// Internal/Blocks/GetStatusMessage
(* ===============================================================================
   FESTO AG & Co. KG, Esslingen - Copyright 2015. All rights reserved.                       
 ---------------------------------------------------------------------------------
 Functionblock:  GetStatusMessage 
 Description:    function to get discription of the status of function block or FPC 
 Version:        V 1.0        
 Composer:       Benjamin Kilgus
 Last Update:    10.04.2014                                                                          
------------------------------------------------------------------------------- *)
{library private}
(* ----------------------------------------------------------------------------
Date        Name            	Activity                                                                              
10.04.2014	Benjamin Kilgus     created
=============================================================================== *)
{library public}

FUNCTION GetStatusMessage : STRING

VAR_INPUT
  StatusIn   	: DT_FML_STATUS;
END_VAR

VAR
  StatusStringCat  	: STRING;
  StatusStringID  	: STRING;
END_VAR

(* ===== logic part ================================================= *)
 // get category string 
 CASE StatusIn.Cat OF
	 
 	FML_no_category:
		StatusStringCat := '';
		// get ID string 
		CASE StatusIn.ID OF
			 0:     StatusStringID := 'no error';
			 ELSE   StatusStringID := 'unknown number';
		END_CASE

		 
	FML_function_block:	
		StatusStringCat := 'FB: ';
		// get ID string 
	  	CASE StatusIn.ID OF
			 0:     StatusStringID := 'no error';
			 1:     StatusStringID := 'initialization is active';
			 2:     StatusStringID := 'function block is busy';
			10:     StatusStringID := 'other FPC function block is active';
			20:     StatusStringID := 'timeout of function block';
			30:     StatusStringID := 'device type is not valid';
			40:     StatusStringID := 'wrong access value';
			50:     StatusStringID := 'pointer to zero';
			51:     StatusStringID := 'pointer wrong size';
			60:     StatusStringID := 'FHPP+ data configuration not valid';
			ELSE 	StatusStringID := 'unknown number';
		END_CASE
		
		
	FML_reserved:
		StatusStringCat := 'reserved: ';

	FML_parameter_transfer:
		StatusStringCat	:= 'FPC: ';
		// get ID string 
	  	CASE StatusIn.ID OF
			 0:      StatusStringID := 'non-permitted PNU';
			 1:      StatusStringID := 'parameter is read only';
			 2:      StatusStringID := 'lower or upper limit value exceeded';
			 3:      StatusStringID := 'wrong subindex';
			 4:      StatusStringID := 'no array';
			 5:      StatusStringID := 'incorrect data type';
			 6:      StatusStringID := 'setting not permitted (only reset allowed)';
			 7:      StatusStringID := 'describing element cannot be modified';
			 8:      StatusStringID := 'PPO-Write requested in IR does not exist';
			 9:      StatusStringID := 'description data do not exist';
			10:      StatusStringID := 'access group incorrect';
			11:      StatusStringID := 'no control rights';
			12:      StatusStringID := 'password incorrect';
			13:      StatusStringID := 'text not readable in cyclic exchange';
			14:      StatusStringID := 'name not readable in cyclic exchange';
			15:      StatusStringID := 'text array does not exist';
			16:      StatusStringID := 'PPO-Write missing';
			17:      StatusStringID := 'order cannot be processed because of operating status';
			18:      StatusStringID := 'other Errors';
			19:      StatusStringID := 'date not readable in cyclic exchange';
			20:      StatusStringID := 'non-permitted value';
			22:      StatusStringID := 'non-permitted Attributes, number of elements, PNU or IND';
			23:      StatusStringID := 'write request: non-permitted format';
			24:      StatusStringID := 'write request: Number of values not permitted';
			25..100: StatusStringID := 'reserved for PROFIBUS';
			101:     StatusStringID := 'ReqID is not supported';
			102:     StatusStringID := 'parameter is write only';
			103..255:StatusStringID := 'reserved for Festo';
			
			//FILETRANSFER
			1001: 	StatusStringID := 'wrong sequence number';
			1002: 	StatusStringID := 'timeout between two packets';
			1003: 	StatusStringID := 'wrong packet format';
			1004: 	StatusStringID := 'false instruction';
			1005: 	StatusStringID := 'read error';
			1006:	StatusStringID := 'write error';
			1007:	StatusStringID := 'data volume is not correct';
			1008: 	StatusStringID := 'parameterfile error';
			1009: 	StatusStringID := 'fault not receipt';
			1010: 	StatusStringID := 'timeout';
			1011: 	StatusStringID := 'file open error';
			1012: 	StatusStringID := 'file close error';
			1013: 	StatusStringID := 'file delete error';
			1014: 	StatusStringID := 'directory create error';
			1015: 	StatusStringID := 'file not exist';
			1016: 	StatusStringID := 'file read error';
			1017: 	StatusStringID := 'get size error';
			1018: 	StatusStringID := 'file write error';
			1019:	StatusStringID := 'no or double direction selected';
			1020:	StatusStringID := 'filename is empty';
			1021:	StatusStringID := 'size of parameterfile too short/long';
			1022:	StatusStringID := 'parameterfile is not complete';
			
			ELSE 	StatusStringID := 'unknown number';
		END_CASE
			
	ELSE
		StatusStringCat := 'unknown status category';
 END_CASE

 
 GetStatusMessage := CONCAT(StatusStringCat, StatusStringID);  // Return the resulting string
 
(* ===== end of function ================================== *)

END_FUNCTION

// Blocks/FML_Read
(* ============================================================================
   FESTO AG & Co. KG, Esslingen - Copyright (c) 2015. All rights reserved.                       

 Functionblock:  FML_Read
 Description:    function block to read the input data from the controller
 Version:        V3.5.7.21        
 Composer:       chmm
 Date:           13.11.2017                                                                          
------------------------------------------------------------------------------- *)
{library private}
(* ----------------------------------------------------------------------------
Date        Name             	Activity                                                                              
22.06.2015	Christian Hammer	created
13.11.2017	Christian Hammer	added SFC-DC and MTR-DCI controller
=============================================================================== *)
{library public}


FUNCTION_BLOCK FML_Read

VAR_IN_OUT
	FML_REF					: DT_FML_REF; 						// structure of the parameter to control and parametrize the motorcontroller
END_VAR

VAR_INPUT
	DeviceType				: E_FML_DEVICE_TYPE; 				// type of the controller
	Modbus					: BOOL;								// 1 = modbus is using / 0 = other fieldbus is using
	HighByteFirst			: BOOL;								// byteorder (1 = high byte first)
	FPC_active				: BOOL;								// ParameterChannel (FPC) in use
	PlcConfigFHPP_PLUS_IN	: UDINT;							// plc configuration code (is displayed in the Festo Configuration Tool (FCT))
	
	FHPP_Source				: ARRAY [0..7] OF BYTE;				// input FHPP Data (from controller)
	FPC_Source				: ARRAY [0..7] OF BYTE;				// input FPC Data (from controller)
	FHPP_PLUS_Source1		: ARRAY [0..7] OF BYTE;				// first 8 bytes of FHPP+ input data (from controller)
	FHPP_PLUS_Source2		: ARRAY [0..7] OF BYTE;				// second 8 bytes of FHPP+ input data (from controller)
	FHPP_PLUS_Source3		: ARRAY [0..7] OF BYTE;				// third 8 bytes of FHPP+ input data (from controller)
END_VAR

VAR_OUTPUT
	Error					: BOOL;								// transmission fault
	Status          		: DT_FML_STATUS;     				// return value of function block
END_VAR

VAR
	FHPP_Read				: FHPP_Read;						// function block read FHPP data
	FPC_Read				: FPC_Read;							// function block read FPC data
	FHPP_PLUS_Read			: FHPP_PLUS_Read;					// function block read FHPP+ data
END_VAR

// function block (FB) is busy
Status.Err:=FALSE; Status.Cat:=FML_function_block; Status.ID:=FML_fb_busy;

// check and set DeviceType of the controller
IF DeviceType = CMMO_ST OR DeviceType = EMCA_EC OR DeviceType = CMMP_AS OR DeviceType = CMMS_AS OR DeviceType = CMMS_ST OR DeviceType = CMMD_AS OR DeviceType = SFC_DC OR DeviceType = MTR_DCI THEN  
	FML_REF.DeviceType	:= DeviceType;
ELSE
	Status.Err:=TRUE; Status.Cat:=FML_function_block; Status.ID:=FML_wrong_device;
END_IF

// set type of bus and byteorder
FML_REF.Modbus			:= Modbus;
FML_REF.HighByteFirst	:= HighByteFirst;

// mode of the parameter channel (in use or not)
FML_REF.FPC_active		:= FPC_active;

// reading and mapping of FHPP bus data 
FHPP_Read(
	FML_REF				:= FML_REF,
	FHPP_Source			:= FHPP_Source);
		
// if parameter-channel (FPC) is activated - reading and mapping of FPC bus data	
IF FML_REF.FPC_active THEN
	FPC_Read(
		FML_REF			:= FML_REF,
		FPC_Source		:= FPC_Source);
END_IF

IF (PlcConfigFHPP_PLUS_IN<>0) AND (Status.Err = FALSE) THEN
	FHPP_PLUS_Read(
		FML_REF					:= FML_REF,
		PlcConfigFHPP_PLUS_IN	:= PlcConfigFHPP_PLUS_IN,
		FHPP_PLUS_Source1		:= FHPP_PLUS_Source1,
		FHPP_PLUS_Source2		:= FHPP_PLUS_Source2,
		FHPP_PLUS_Source3		:= FHPP_PLUS_Source3,
		Status					=> Status);		
END_IF	
	
IF (Status.Err = FALSE) THEN
	// reading done - no error
	Status.Err:=FALSE; Status.Cat:=FML_no_category; Status.ID:=FML_no_error;
END_IF	

Status.Msg						:= GetStatusMessage(Status);
Error							:= Status.Err;

(* ===== end of function block ============================= *)

END_FUNCTION_BLOCK

// Internal/Blocks/ReadWriteData/FHPP_Read
(* ===============================================================================
   FESTO AG & Co. KG, Esslingen - Copyright 2015. All rights reserved.                       
 ---------------------------------------------------------------------------------
 Functionblock:  FHPP_Read  
 Description:    function block to read an mapp the FHPP data from the controller
 Version:        V 3.5.4.4        
 Composer:       chmm 
 Last Update:    22.06.2015                                                                           
------------------------------------------------------------------------------- *)
{library private}
(* ----------------------------------------------------------------------------
Date        Name            	Activity                                                                              
22.06.2015	Christian Hammer	created
=============================================================================== *)
{library public}

FUNCTION_BLOCK FHPP_Read

VAR_IN_OUT
	FML_REF			: DT_FML_REF;						// structure of the parameter to control and parametrize the motorcontroller
END_VAR

VAR_INPUT
	FHPP_Source		: ARRAY [0..7] OF BYTE;				// input FHPP data (from controller)
END_VAR

VAR
	pFHPP_DATA_IN	: POINTER TO ARRAY[0..7] OF BYTE;	// pointer to FHPP data
END_VAR

(***********************************************************************************************************************************************
*********** INPUT FHPP DATA ********************************************************************************************************************
***********************************************************************************************************************************************)

pFHPP_DATA_IN				:= ADR(FML_REF.FHPP.IN);

IF FML_REF.Modbus THEN				// modbus word swapping
	pFHPP_DATA_IN^[0]		:= FHPP_Source[1]; 
	pFHPP_DATA_IN^[1]		:= FHPP_Source[0]; 
	pFHPP_DATA_IN^[2]		:= FHPP_Source[3]; 
	pFHPP_DATA_IN^[3]		:= FHPP_Source[2];
	IF FML_REF.HighByteFirst THEN	// high byte first (actual value2)
		pFHPP_DATA_IN^[4]	:= FHPP_Source[6]; 
		pFHPP_DATA_IN^[5] 	:= FHPP_Source[7]; 
		pFHPP_DATA_IN^[6] 	:= FHPP_Source[4]; 
		pFHPP_DATA_IN^[7] 	:= FHPP_Source[5];
	ELSE							// low byte first (actual value2)
		pFHPP_DATA_IN^[4]	:= FHPP_Source[5]; 
		pFHPP_DATA_IN^[5] 	:= FHPP_Source[4]; 
		pFHPP_DATA_IN^[6] 	:= FHPP_Source[7]; 
		pFHPP_DATA_IN^[7] 	:= FHPP_Source[6];
	END_IF

ELSE								// normal fieldbus: copy only
	pFHPP_DATA_IN^[0]		:= FHPP_Source[0]; 
	pFHPP_DATA_IN^[1]		:= FHPP_Source[1]; 
	pFHPP_DATA_IN^[2]		:= FHPP_Source[2]; 
	pFHPP_DATA_IN^[3]		:= FHPP_Source[3]; 
	IF FML_REF.HighByteFirst THEN	// high byte first (actual value2)
		pFHPP_DATA_IN^[4]	:= FHPP_Source[7]; 
		pFHPP_DATA_IN^[5] 	:= FHPP_Source[6]; 
		pFHPP_DATA_IN^[6] 	:= FHPP_Source[5]; 
		pFHPP_DATA_IN^[7] 	:= FHPP_Source[4];
	ELSE							// low byte first (actual value2)
		pFHPP_DATA_IN^[4]	:= FHPP_Source[4]; 
		pFHPP_DATA_IN^[5] 	:= FHPP_Source[5]; 
		pFHPP_DATA_IN^[6] 	:= FHPP_Source[6]; 
		pFHPP_DATA_IN^[7] 	:= FHPP_Source[7];
	END_IF
END_IF

(* ===== end of function block ============================= *)

END_FUNCTION_BLOCK

// Internal/Blocks/ReadWriteData/FPC_Read
(* ===============================================================================
   FESTO AG & Co. KG, Esslingen - Copyright 2015. All rights reserved.                       
 ---------------------------------------------------------------------------------
 Functionblock:  FPC_Read  
 Description:    function block to read an mapp the FPC data from the controller
 Version:        V 3.5.7.21        
 Composer:       chmm 
 Last Update:    20.11.2017                                                                           
------------------------------------------------------------------------------- *)
{library private}
(* ----------------------------------------------------------------------------
Date        Name            	Activity                                                                              
22.06.2015	Christian Hammer	created
20.11.2017	Christian Hammer	ResponseID´s for SFC-DC and MTR-DCI added
=============================================================================== *)
{library public}

FUNCTION_BLOCK FPC_Read

VAR_IN_OUT
	FML_REF			: DT_FML_REF;						// structure of the parameter to control and parametrize the motorcontroller
END_VAR	

VAR_INPUT
	FPC_Source		: ARRAY [0..7] OF BYTE;				// input FPC data (from controller)
END_VAR

VAR
	pFPC_DATA_IN	: POINTER TO ARRAY[0..7] OF BYTE;	// pointer to FPC data
	pFML_Ref_FPC_In	: POINTER TO ARRAY[0..7] OF BYTE;	// pointer to FML-Ref-FPC.In for copying paramter files or firmware files
	RespID			: INT;
END_VAR

(***********************************************************************************************************************************************
*********** INPUT FPC DATA *********************************************************************************************************************
***********************************************************************************************************************************************)

pFPC_DATA_IN				:= ADR(FML_REF.FPC.IN);

IF FML_REF.Modbus THEN				// modbus word swapping
	pFPC_DATA_IN^[0]		:= FPC_Source[1]; 
	pFPC_DATA_IN^[1]		:= FPC_Source[0]; 
	IF FML_REF.HighByteFirst THEN	// high bytes first (ParID and value)
		pFPC_DATA_IN^[2]	:= FPC_Source[2]; 
		pFPC_DATA_IN^[3]	:= FPC_Source[3];
		pFPC_DATA_IN^[4]	:= FPC_Source[6]; 
		pFPC_DATA_IN^[5] 	:= FPC_Source[7]; 
		pFPC_DATA_IN^[6] 	:= FPC_Source[4]; 
		pFPC_DATA_IN^[7] 	:= FPC_Source[5];
	ELSE							// low bytes first (ParID and value)
		pFPC_DATA_IN^[2]	:= FPC_Source[3]; 
		pFPC_DATA_IN^[3]	:= FPC_Source[2];
		pFPC_DATA_IN^[4]	:= FPC_Source[5]; 
		pFPC_DATA_IN^[5] 	:= FPC_Source[4]; 
		pFPC_DATA_IN^[6] 	:= FPC_Source[7]; 
		pFPC_DATA_IN^[7] 	:= FPC_Source[6];
	END_IF

ELSE								//normal fieldbus: copy only
	pFPC_DATA_IN^[0]		:= FPC_Source[0]; 
	pFPC_DATA_IN^[1]		:= FPC_Source[1];
	IF FML_REF.HighByteFirst THEN	// high byte first (ParID and value)
		pFPC_DATA_IN^[2]	:= FPC_Source[3]; 
		pFPC_DATA_IN^[3]	:= FPC_Source[2];
		pFPC_DATA_IN^[4]	:= FPC_Source[7]; 
		pFPC_DATA_IN^[5] 	:= FPC_Source[6]; 
		pFPC_DATA_IN^[6] 	:= FPC_Source[5]; 
		pFPC_DATA_IN^[7] 	:= FPC_Source[4];	
	ELSE 							// low bytes first (ParID and value)
		pFPC_DATA_IN^[2]	:= FPC_Source[2]; 
		pFPC_DATA_IN^[3]	:= FPC_Source[3];
		pFPC_DATA_IN^[4]	:= FPC_Source[4]; 
		pFPC_DATA_IN^[5] 	:= FPC_Source[5]; 
		pFPC_DATA_IN^[6] 	:= FPC_Source[6]; 
		pFPC_DATA_IN^[7] 	:= FPC_Source[7];
	END_IF	
END_IF



(*-----------------------------------------------------------
     assignment of the input data (stateword)
------------------------------------------------------------*)
(* byte 1 FPCS *)
FML_REF.FPCS_Modus 				:= SHR((FML_REF.FPC.IN.ModeAK AND 2#11110000),4);

(*-----------------------------------------------------------
     decoding of EFPC modus
------------------------------------------------------------*)
CASE FML_REF.FPCS_Modus OF
	1,2,3:(* FPCS_Modus 1=PNU extended; 2= internal data object; 3=CAN objects *)

	(*
	|-------- byte 1 ------|- byte 2 -|---------- byte 3..4 ------------------------|- byte 5..8 -|
	| 7  6  5  4 | 3 2 1 0 |          | 15 14 ..                 			 .. 1 0 |             |
	| FPCS mode	 |   AK    | subindex | PNU extended or data object or CAN object	|    value    |
	-----------------------------------------------------------------------------------------------		
		AK:  request identifier (Auftragskennung) *)			
		
		FML_REF.RespID	 		:= (FML_REF.FPC.IN.ModeAK AND 2#00001111);		// FPCS mode (byte 1)	
		FML_REF.ActSubindex 	:= FML_REF.FPC.IN.IND;   						// save subindex (byte 2)		
		FML_REF.ActValue		:= FML_REF.FPC.IN.Value; 						// parameter value (byte 5..8)
		FML_REF.ActPNU 			:= FML_REF.FPC.IN.ParID;						// **PKE/ PNU/ data object/ CAN (byte 3+4)

	4,5:(* FPCS_Modus 4=parameter file; 5=firmware file 
      	|------ byte 1 -----------|-- byte 2 -|--byte 3..8 -----|
	    | 7  6  5  4 | 3  2  1  0 |           | 				|
	    | FPCS Modus |   res      | Packet-ID |  6 Byte Data	|
	    -------------------------------------------------------		
		  packet-ID: -------------- byte 2 ----------
		             | 7    6    5  | 4  3  2  1  0 |
		             | control bits |   sequence-nr |
		             -------------------------------- *)		
		//---- FPCS mode (byte 1) ---- 
		FML_REF.RespID						:= (FML_REF.FPC.IN.ModeAK AND 2#00001111);
		//---- byte 2 packet-ID ----	
		FML_REF.FPCS_Packet.BitSequenceNr 	:= (FML_REF.FPC.IN.IND AND 2#00011111);
		FML_REF.FPCS_Packet.Control			:= SHR((FML_REF.FPC.IN.IND AND 2#11100000),5);
		//---- byte 3..8 data ----	
		pFML_Ref_FPC_In						:= ADR(FML_REF.FPC.IN);			// byte swapping for modbus data
		FML_REF.FPCS_Packet.Data[1]			:= pFML_Ref_FPC_In^[3];  
		FML_REF.FPCS_Packet.Data[2] 		:= pFML_Ref_FPC_In^[2];  
		FML_REF.FPCS_Packet.Data[3] 		:= pFML_Ref_FPC_In^[7];  
		FML_REF.FPCS_Packet.Data[4] 		:= pFML_Ref_FPC_In^[6];  
		FML_REF.FPCS_Packet.Data[5] 		:= pFML_Ref_FPC_In^[5];  
		FML_REF.FPCS_Packet.Data[6] 		:= pFML_Ref_FPC_In^[4]; 
	
	ELSE  (* FPCS_Modus = standard ----
  		|-byte 1 -|- byte 2 -|---------------- byte 3 --------------|- byte 5..8 -|
		|         |          |15 14 13 12| 11|10 9 8 7 6 5 4 3 2 1 0|             |
		|   res   | subindex |     AK    |SPM|        PNU           |   value     |
		---------------------------------------------------------------------------		
			byte 1: reserved
			byte 2: subindex
			AK:     response identifier (Antwortkennung)
			SPM:    NOT used
			PNU:    Parameternummer / parametern umber *)				

		FML_REF.ActSubindex 	:= FML_REF.FPC.IN.IND;  	 // save subindex
		
		(* Byte 3+4 **PKE/ PNU/ data object/ CAN** *)
		FML_REF.ActValue		:= FML_REF.FPC.IN.Value;
		RespID					:= WORD_TO_INT( SHR((INT_TO_WORD(FML_REF.FPC.IN.ParID) AND 2#1111000000000000),12));
		FML_REF.RespID			:= RespID;
		FML_REF.ActPNU 			:= WORD_TO_INT( INT_TO_WORD(FML_REF.FPC.IN.ParID) AND 2#0000011111111111);
		
		(* Byte 5..8 parameter value *)
END_CASE

CASE FML_REF.RespID OF
	
	 0,3:(* No instruction or transmission is activ *)
		FML_REF.Done            := FALSE;
		FML_REF.Err             := FALSE;
		FML_REF.DatatypeRD      := 0;
		FML_REF.ActPNU          := 0;
		FML_REF.ActSubindex     := 0;
		FML_REF.ActValue    	:= 0;
			
	1,4:(* WORD Parameter transmitted *)
		FML_REF.Done            := TRUE;
		FML_REF.Err             := FALSE;
		FML_REF.DatatypeRD      := 2;
	
	2,5:(* DWORD Parameter transmitted *)
		FML_REF.Done            := TRUE;
		FML_REF.Err             := FALSE;
		FML_REF.DatatypeRD      := 4;
			
	7:(* Transmission Err *)
		FML_REF.Done            := TRUE;
		FML_REF.Err             := TRUE;
		FML_REF.DatatypeRD      := 0;
			
	11,12:(* BYTE Parameter transmitted *)
		FML_REF.Done            := TRUE;
		FML_REF.Err             := FALSE;
		FML_REF.DatatypeRD      := 1;
		
	ELSE (* not specified*)
		FML_REF.Done        	:= TRUE;
		FML_REF.Err           	:= TRUE;
		FML_REF.DatatypeRD      := 0;	
END_CASE

(* ===== end of function block ============================= *)

END_FUNCTION_BLOCK

// Blocks/FML_Write
(* ============================================================================
   FESTO AG & Co. KG, Esslingen - Copyright (c) 2015. All rights reserved.                       

 Functionblock:  FML_Write
 Description:    function block to write the output data to the controller
 Version:        V3.5.4.4        
 Composer:       chmm
 Date:           04.09.2015                                                                           
------------------------------------------------------------------------------- *)
{library private}
(* ----------------------------------------------------------------------------
Date        Name             	Activity                                                                              
22.06.2015	Christian Hammer	created	
=============================================================================== *)
{library public}

FUNCTION_BLOCK FML_Write

VAR_IN_OUT
	FML_REF					: DT_FML_REF; 
END_VAR

VAR_INPUT
	PlcConfigFHPP_PLUS_OUT	: UDINT;							// plc configuration code for the FHPP+ output(is displayed in the Festo Configuration Tool (FCT))
END_VAR

VAR_OUTPUT
	FHPP_Target				: ARRAY [0..7] OF BYTE;				// Output FHPP Data (to controller)
	FPC_Target				: ARRAY [0..7] OF BYTE;				// Output FPC Data (to controller)
	FHPP_PLUS_Target1		: ARRAY [0..7] OF BYTE;				// first 8 bytes of FHPP+ output data (to controller)
	FHPP_PLUS_Target2		: ARRAY [0..7] OF BYTE;				// second 8 bytes of FHPP+ output data (to controller)
	FHPP_PLUS_Target3		: ARRAY [0..7] OF BYTE;				// third 8 bytes of FHPP+ output data (to controller)
	Error					: BOOL;								// transmission fault
	Status          		: DT_FML_STATUS;     				// return value of function block
END_VAR

VAR
	FHPP_Write				: FHPP_Write;						// function block write FHPP data
	FPC_Write				: FPC_Write;						// function block write FPC data
	FHPP_PLUS_Write			: FHPP_PLUS_Write;					// function block write FHPP+ data
END_VAR

// function block (FB) is busy
Status.Err:=FALSE; Status.Cat:=FML_function_block; Status.ID:=FML_fb_busy;

// mapping and writeing of FHPP bus data 
FHPP_Write(
	FML_REF		:= FML_REF,
	FHPP_Target	=> FHPP_Target);
		
// if parameter-channel (FPC) is activated - mapping and writeing of FPC bus data	
IF FML_REF.FPC_active THEN
	FPC_Write(
		FML_REF		:= FML_REF,
		FPC_Target	=> FPC_Target);
END_IF

IF PlcConfigFHPP_PLUS_OUT<>0 THEN
	FHPP_PLUS_Write(
		FML_REF					:= FML_REF,
		PlcConfigFHPP_PLUS_OUT	:= PlcConfigFHPP_PLUS_OUT,
		FHPP_PLUS_Target1		=> FHPP_PLUS_Target1,
		FHPP_PLUS_Target2		=> FHPP_PLUS_Target2,
		FHPP_PLUS_Target3		=> FHPP_PLUS_Target3,
		Status					=> Status);
END_IF		

IF Status.Err = FALSE THEN
	// writing done - no error
	Status.Err:=FALSE; Status.Cat:=FML_no_category; Status.ID:=FML_no_error;
END_IF	

Status.Msg				:= GetStatusMessage(Status);
Error					:= Status.Err;

(* ===== end of function block ============================= *)

END_FUNCTION_BLOCK

// Internal/Blocks/ReadWriteData/FHPP_Write
(* ===============================================================================
   FESTO AG & Co. KG, Esslingen - Copyright 2015. All rights reserved.                       
 ---------------------------------------------------------------------------------
 Functionblock:  FHPP_Write  
 Description:    function block to write the FHPP data to the controller
 Version:        V 3.5.4.4        
 Composer:       chmm 
 Last Update:    22.06.2015                                                                           
------------------------------------------------------------------------------- *)
{library private}
(* ----------------------------------------------------------------------------
Date        Name            	Activity                                                                              
22.06.2015	Christian Hammer	created
=============================================================================== *)
{library public}

FUNCTION_BLOCK FHPP_Write

VAR_IN_OUT
	FML_REF			: DT_FML_REF; 						// structure of the parameter to control and parametrize the motorcontroller
END_VAR

VAR_OUTPUT
	FHPP_Target		: ARRAY [0..7] OF BYTE;				// output FHPP data
END_VAR

VAR
	pFHPP_DATA_OUT	: POINTER TO ARRAY[0..7] OF BYTE;	// pointer to FHPP data
END_VAR

(***********************************************************************************************************************************************
*********** OUTPUT FHPP DATA *******************************************************************************************************************
***********************************************************************************************************************************************)

pFHPP_DATA_OUT				:= ADR(FML_REF.FHPP.OUT);

IF FML_REF.Modbus THEN				// modbus word swapping
	FHPP_Target[0]			:= pFHPP_DATA_OUT^[1];
	FHPP_Target[1]			:= pFHPP_DATA_OUT^[0];
	FHPP_Target[2]			:= pFHPP_DATA_OUT^[3];
	FHPP_Target[3]			:= pFHPP_DATA_OUT^[2];
	IF FML_REF.HighByteFirst THEN	// high byte first (actual value2)
		FHPP_Target[4]		:= pFHPP_DATA_OUT^[6];
		FHPP_Target[5]		:= pFHPP_DATA_OUT^[7];
		FHPP_Target[6]		:= pFHPP_DATA_OUT^[4];
		FHPP_Target[7]		:= pFHPP_DATA_OUT^[5];
	ELSE							// low byte first (actual value2)
		FHPP_Target[4]		:= pFHPP_DATA_OUT^[5];
		FHPP_Target[5]		:= pFHPP_DATA_OUT^[4];
		FHPP_Target[6]		:= pFHPP_DATA_OUT^[7];
		FHPP_Target[7]		:= pFHPP_DATA_OUT^[6];
	END_IF	
	
ELSE								//normal fieldbus: copy only
	FHPP_Target[0]			:= pFHPP_DATA_OUT^[0];
	FHPP_Target[1]			:= pFHPP_DATA_OUT^[1];
	FHPP_Target[2]			:= pFHPP_DATA_OUT^[2];
	FHPP_Target[3]			:= pFHPP_DATA_OUT^[3];
	IF FML_REF.HighByteFirst THEN	// high byte first (actual value2)
		FHPP_Target[4]		:= pFHPP_DATA_OUT^[7];
		FHPP_Target[5]		:= pFHPP_DATA_OUT^[6];
		FHPP_Target[6]		:= pFHPP_DATA_OUT^[5];
		FHPP_Target[7]		:= pFHPP_DATA_OUT^[4];
	ELSE							// low byte first (actual value2)
		FHPP_Target[4]		:= pFHPP_DATA_OUT^[4];
		FHPP_Target[5]		:= pFHPP_DATA_OUT^[5];
		FHPP_Target[6]		:= pFHPP_DATA_OUT^[6];
		FHPP_Target[7]		:= pFHPP_DATA_OUT^[7];
	END_IF	
END_IF

(* ===== end of function block ============================= *)

END_FUNCTION_BLOCK

// Internal/Blocks/ReadWriteData/FPC_Write
(* ===============================================================================
   FESTO AG & Co. KG, Esslingen - Copyright 2015. All rights reserved.                       
 ---------------------------------------------------------------------------------
 Functionblock:  FPC_Write  
 Description:    function block to write the FPC data to the controller
 Version:        V 3.5.7.21        
 Composer:       chmm 
 Last Update:    20.11.2017                                                                           
------------------------------------------------------------------------------- *)
{library private}
(* ----------------------------------------------------------------------------
Date        Name            	Activity                                                                              
22.06.2015	Christian Hammer	created
20.11.2017	Christian Hammer	SFC-DC and MTR-DCI added
=============================================================================== *)
{library public}

FUNCTION_BLOCK FPC_Write

VAR_IN_OUT
	FML_REF				: DT_FML_REF; 						// structure of the parameter to control and parametrize the motorcontroller
END_VAR

VAR_OUTPUT
	FPC_Target			: ARRAY [0..7] OF BYTE;				// output FPC data
END_VAR

VAR
	pFPC_DATA_OUT		: POINTER TO ARRAY[0..7] OF BYTE;	// pointer to FPC data  
	pFML_Ref_FPC_Out	: POINTER TO ARRAY[0..7] OF BYTE;	// pointer to FML-Ref-FPC.Out for copying paramter files or firmware files
	Req_Identifier		: WORD;
END_VAR

(*-----------------------------------------------------------
     assignment of the output data (control word)
------------------------------------------------------------*)
IF FML_REF.DeviceType = SFC_DC OR FML_REF.DeviceType = MTR_DCI THEN							(* SFC-DC or MTR-DCI *)
	IF FML_REF.ReqID = FML_FPC_REQ_write_array_dword THEN
		IF FML_REF.Subindex > 0 THEN
     		CASE FML_REF.DatatypeWR OF			(** write array **)
      			1:		FML_REF.ReqID	:= 12;		// array of byte
        		2:		FML_REF.ReqID	:= 7;		// array of word
        		4:		FML_REF.ReqID	:= 8;		// array of dword
				ELSE	FML_REF.ReqID	:= 8;		// array of dword	
     		 END_CASE
		
		ELSIF FML_REF.Subindex = 0 THEN			(** write single parameter **)
      		CASE FML_REF.DatatypeWR OF
        		1:		FML_REF.ReqID	:= 11;   	// array of byte
        		2:		FML_REF.ReqID	:= 2;	  	// array of word
        		4:		FML_REF.ReqID	:= 3;	   	// array of dword
				ELSE	FML_REF.ReqID	:= 3;	   	// array of dword
      		END_CASE
			
		ELSE
			FML_REF.ReqID				:= 0;	(** do nothing **)
    	END_IF
		
	ELSIF FML_REF.ReqID = FML_FPC_REQ_read_array THEN
		IF FML_REF.Subindex > 0 THEN  			(** read array **)
      		FML_REF.ReqID 				:= 6;
   		
		ELSIF FML_REF.Subindex	= 0 THEN  		(** read single parameter **)
      		FML_REF.ReqID				:= 1;
    	
		ELSE
			FML_REF.ReqID				:= 0;	(** do nothing **)
    	END_IF
	END_IF
END_IF


CASE FML_REF.FPCC_Modus OF 
	1,2,3:(* FPCC_Modus 1=PNU extended; 2= internal data object; 3=CAN objects 
		---------- Byte 1 ------|-Byte 2 |-------------- byte 3..4 --------------------	|- byte 5..8 -|
		|  8 7 6 5 4  | 3 2 1 0 |        |15 14 13 12 11 10 9 8 7 6 5 4 3 2 1 0			|             |
		| FPCS modus  |   AK    |subindex|  PNU extended or data object or CAN object  	|   value     |
		----------------------------------------------------------------------------------------------	
		AK:  request identifier (Auftragskennung) *)		
		
		FML_REF.FPC.OUT.ModeAK			:= (SHL(DINT_TO_BYTE(FML_REF.FPCC_Modus),4) OR INT_TO_BYTE(FML_REF.ReqID));	// byte 1
		FML_REF.FPC.OUT.IND				:= DINT_TO_BYTE(FML_REF.Subindex);											// byte 2 subindex 
		
		FML_REF.FPC.OUT.ParID			:= FML_REF.PNU;      														// byte 3+4 	
		FML_REF.FPC.OUT.Value			:= FML_REF.Value;  															// byte 5..8
    
	4,5:(* FPCC_Modus 4=parameter file; 5=firmware file 	
		|---------- byte 1 --------|-- byte 2 --|-- byte 3..8 ---|
		| 7  6  5  4  | 3  2  1  0 |            | 				 |
		|	FPCC modus |   res      | packet-ID  |  6 byte data	 |
		---------------------------------------------------------		
		Packet-ID:  | 7    6    5  | 4  3  2  1  0  |
		            | control bits |  sequence-nr   |
		            --------------------------------- *)				
		//---- byte 1 ----
		FML_REF.FPC.OUT.ModeAK			:= (SHL (DINT_TO_BYTE(FML_REF.FPCC_Modus),4)OR (INT_TO_BYTE(FML_REF.ReqID)));
		//----byte 2 packet-ID ----	
		FML_REF.FPC.OUT.IND 			:= (SHL (INT_TO_BYTE(FML_REF.FPCC_Packet.Control),5) OR (INT_TO_BYTE(FML_REF.FPCC_Packet.BitSequenceNr) AND 16#1F ));
		//---- byte 3..8 data ----
		pFML_Ref_FPC_Out				:= ADR(FML_REF.FPC.OUT);
		pFML_Ref_FPC_Out^[2]			:= FML_REF.FPCC_Packet.Data[2];			// byte swapping for modbus data 
		pFML_Ref_FPC_Out^[3]			:= FML_REF.FPCC_Packet.Data[1];	
		pFML_Ref_FPC_Out^[4]			:= FML_REF.FPCC_Packet.Data[6];	
		pFML_Ref_FPC_Out^[5]			:= FML_REF.FPCC_Packet.Data[5];	
		pFML_Ref_FPC_Out^[6]			:= FML_REF.FPCC_Packet.Data[4];	
		pFML_Ref_FPC_Out^[7]			:= FML_REF.FPCC_Packet.Data[3];
		
	ELSE (* FPCC_Modus standard 
		| byte 1 -|- byte 2 -|---------------- byte 3 --------------|- byte 5..8 -|
		|         |          |15 14 13 12| 11|10 9 8 7 6 5 4 3 2 1 0|             |
		|   res   | subindex |     AK    |SPM|        PNU           |   value     |
		---------------------------------------------------------------------------		
			AK:  response identifier (Antwortkennung)
			SPM: NOT used
			PNU: Parameternummer / parameter number *)				
		
		FML_REF.FPC.OUT.ModeAK 			:= 0;               				// byte 1 
		FML_REF.FPC.OUT.IND 			:= DINT_TO_BYTE(FML_REF.Subindex); 	// byte 2 subindex
		//---- Byte 3+4 ---- 
		FML_REF.FPC.OUT.ParID			:= WORD_TO_INT(SHL((INT_TO_WORD(FML_REF.ReqID)),12) OR (INT_TO_WORD(FML_REF.PNU) AND 16#07_FF));
		FML_REF.FPC.OUT.Value 			:= FML_REF.Value;
END_CASE



(***********************************************************************************************************************************************
*********** OUTPUT FPC DATA ********************************************************************************************************************
***********************************************************************************************************************************************)

pFPC_DATA_OUT				:= ADR(FML_REF.FPC.OUT);

IF FML_REF.Modbus THEN				// modbus word swapping
	FPC_Target[0]			:= pFPC_DATA_OUT^[1];
	FPC_Target[1]			:= pFPC_DATA_OUT^[0];
	IF FML_REF.HighByteFirst THEN	// high byte first (ParID and value)
		FPC_Target[2]		:= pFPC_DATA_OUT^[2];
		FPC_Target[3]		:= pFPC_DATA_OUT^[3];
		FPC_Target[4]		:= pFPC_DATA_OUT^[6];
		FPC_Target[5]		:= pFPC_DATA_OUT^[7];
		FPC_Target[6]		:= pFPC_DATA_OUT^[4];
		FPC_Target[7]		:= pFPC_DATA_OUT^[5];
	ELSE							// low byte first (ParID and value)
		FPC_Target[2]		:= pFPC_DATA_OUT^[3];
		FPC_Target[3]		:= pFPC_DATA_OUT^[2];
		FPC_Target[4]		:= pFPC_DATA_OUT^[5];
		FPC_Target[5]		:= pFPC_DATA_OUT^[4];
		FPC_Target[6]		:= pFPC_DATA_OUT^[7];
		FPC_Target[7]		:= pFPC_DATA_OUT^[6];
	END_IF	
	
ELSE								// normal fieldbus: copy only
	FPC_Target[0]			:= pFPC_DATA_OUT^[0];
	FPC_Target[1]			:= pFPC_DATA_OUT^[1];
	IF FML_REF.HighByteFirst THEN	// high byte first (ParID and value)
		FPC_Target[2]		:= pFPC_DATA_OUT^[3];
		FPC_Target[3]		:= pFPC_DATA_OUT^[2];		
		FPC_Target[4]		:= pFPC_DATA_OUT^[7];
		FPC_Target[5]		:= pFPC_DATA_OUT^[6];
		FPC_Target[6]		:= pFPC_DATA_OUT^[5];
		FPC_Target[7]		:= pFPC_DATA_OUT^[4];
	ELSE							// low byte first (ParID and value)
		FPC_Target[2]		:= pFPC_DATA_OUT^[2];
		FPC_Target[3]		:= pFPC_DATA_OUT^[3];
		FPC_Target[4]		:= pFPC_DATA_OUT^[4];
		FPC_Target[5]		:= pFPC_DATA_OUT^[5];
		FPC_Target[6]		:= pFPC_DATA_OUT^[6];
		FPC_Target[7]		:= pFPC_DATA_OUT^[7];
	END_IF	
END_IF

(* ===== end of function block ============================= *)

END_FUNCTION_BLOCK

// Internal/Blocks/ReadWriteData/FHPP_PLUS_Write
(* ===============================================================================
   FESTO AG & Co. KG, Esslingen - Copyright 2015. All rights reserved.                       
 ---------------------------------------------------------------------------------
 Functionblock:  FHPP_PLUS_Write  
 Description:    function block to write the FHPP+ data to the controller
 Version:        V 3.5.4.4        
 Composer:       chmm 
 Last Update:    19.08.2015                                                                           
------------------------------------------------------------------------------- *)
{library private}
(* ----------------------------------------------------------------------------
Date        Name            	Activity                                                                              
19.08.2015	Christian Hammer	created
=============================================================================== *)
{library public}

FUNCTION_BLOCK FHPP_PLUS_Write

VAR_IN_OUT
	FML_REF					: DT_FML_REF;						// structure of the parameter to control and parametrize the motorcontroller
END_VAR	

VAR_INPUT	
	PlcConfigFHPP_PLUS_OUT	: UDINT;							// plc configuration code for the FHPP+ output (is displayed in the Festo Configuration Tool (FCT))
END_VAR

VAR_OUTPUT
	FHPP_PLUS_Target1		: ARRAY [0..7] OF BYTE;				// first 8 bytes of FHPP+ output data (to controller)
	FHPP_PLUS_Target2		: ARRAY [0..7] OF BYTE;				// second 8 bytes of FHPP+ output data (to controller)
	FHPP_PLUS_Target3		: ARRAY [0..7] OF BYTE;				// third 8 bytes of FHPP+ output data (to controller)
	Status          		: DT_FML_STATUS; 					// return value of function block	
END_VAR

VAR
	FHPP_PLUS_DATA_OUT		: ARRAY[0..23] OF BYTE;				// intern variable to buffer the FHPP+ output data
	pFHPP_PLUS_DATA_OUT		: POINTER TO ARRAY[0..23] OF BYTE;	// pointer to copy the FHPP+ data from the FML_REF into the intern buffer variable - FHPP_PLUS_DATA_OUT
	pFHPP_PLUS_Object		: POINTER TO ARRAY[0..9] OF DINT;	// pointer to copy the FHPP+ data from the FML_REF into the intern buffer variable - FHPP_PLUS_DATA_OUT
	pDataArray				: POINTER TO ARRAY[0..7] OF BYTE;	// pointer to copy the the intern buffer variable (FHPP_PLUS_DATA_OUT) to the bus (to the controller)
	
	stConfigFHPP_PLUS		: STRING[9];						// string with the plc configuration code for the FHPP+ output(is displayed in the Festo Configuration Tool (FCT))
	iCount					: INT;								// counter variable for the loop
	iAddress				: INT;								// counter variable for address of the pointer
	iObject					: INT;								// counter variable for FHPP+ objects in FML_REF
END_VAR

(***********************************************************************************************************************************************
*********** OUTPUT FHPP+ DATA ******************************************************************************************************************
***********************************************************************************************************************************************)

Status.Err:=FALSE; Status.Cat:=FML_function_block; Status.ID:=FML_init_active;

// inizialize the variables
iAddress			:= 0;
iObject				:= 0;
iCount				:= 0;

// inizialize the pointer
pFHPP_PLUS_DATA_OUT	:= ADR(FHPP_PLUS_DATA_OUT);
pFHPP_PLUS_Object	:= ADR(FML_REF.FHPP_PLUS.OUT);

// change PLC-Config from FCT (is a INT) into a string
stConfigFHPP_PLUS	:= UDINT_TO_STRING(PlcConfigFHPP_PLUS_OUT);

Status.Err:=FALSE; Status.Cat:=FML_function_block; Status.ID:=FML_fb_busy;

// FOR loop to copy the intern FHPP+ objects to the bus output data (to the controller)
FOR (iCount := 0) TO 9 BY 1 DO

	// read the PLC-Config string from FCT to copy the right number of bytes to the bus output data
	CASE stConfigFHPP_PLUS[iCount] OF
		
		49:	//ascii code for '1'	--> the size of the output data is 8 BITs --> copy the FHPP+ object into one BYTE
			pFHPP_PLUS_DATA_OUT^[iAddress]	:= DINT_TO_BYTE(pFHPP_PLUS_Object^[iObject]);
			iAddress						:= iAddress + 1;		// increment the counter variable for address of the pointer in increments of 1
			
			
		50:	//ascii code for '2'	--> the size of the output data is 16 BITs --> copy the FHPP+ object into two BYTEs
			IF FML_REF.HighByteFirst THEN	// byteorder = high byte first 
				pFHPP_PLUS_DATA_OUT^[iAddress+1]:= DINT_TO_BYTE(pFHPP_PLUS_Object^[iObject]);
				pFHPP_PLUS_DATA_OUT^[iAddress]	:= DINT_TO_BYTE(SHR(pFHPP_PLUS_Object^[iObject],8));
				
			ELSE							// byteorder = low byte first 
				pFHPP_PLUS_DATA_OUT^[iAddress]	:= DINT_TO_BYTE(pFHPP_PLUS_Object^[iObject]);
				pFHPP_PLUS_DATA_OUT^[iAddress+1]:= DINT_TO_BYTE(SHR(pFHPP_PLUS_Object^[iObject],8));
			END_IF	
			iAddress							:= iAddress + 2;	// increment the counter variable for address of the pointer in increments of 2
		
			
		52:	//ascii code for '4'	--> the size of the output data is 32 BITs --> copy the FHPP+ object into four BYTEs
			IF FML_REF.HighByteFirst THEN	// byteorder = high byte first 
				pFHPP_PLUS_DATA_OUT^[iAddress+3]:= DINT_TO_BYTE(pFHPP_PLUS_Object^[iObject]);
				pFHPP_PLUS_DATA_OUT^[iAddress+2]:= DINT_TO_BYTE(SHR(pFHPP_PLUS_Object^[iObject],8));
				pFHPP_PLUS_DATA_OUT^[iAddress+1]:= DINT_TO_BYTE(SHR(pFHPP_PLUS_Object^[iObject],16));
				pFHPP_PLUS_DATA_OUT^[iAddress]	:= DINT_TO_BYTE(SHR(pFHPP_PLUS_Object^[iObject],24));
				
			ELSE							// byteorder = low byte first
				pFHPP_PLUS_DATA_OUT^[iAddress]	:= DINT_TO_BYTE(pFHPP_PLUS_Object^[iObject]);
				pFHPP_PLUS_DATA_OUT^[iAddress+1]:= DINT_TO_BYTE(SHR(pFHPP_PLUS_Object^[iObject],8));
				pFHPP_PLUS_DATA_OUT^[iAddress+2]:= DINT_TO_BYTE(SHR(pFHPP_PLUS_Object^[iObject],16));
				pFHPP_PLUS_DATA_OUT^[iAddress+3]:= DINT_TO_BYTE(SHR(pFHPP_PLUS_Object^[iObject],24));
			END_IF	
			iAddress							:= iAddress + 4;	// increment the counter variable for address of the pointer in increments of 4
			
			
		48, 51, 53, 54, 55, 56, 57:	//ascii code for '0', '3', '5', '6', '7', '8', '9' --> wrong number is in the plc configuration code for the FHPP+ input(is displayed in the Festo Configuration Tool (FCT))
			Status.Err:=TRUE; Status.Cat:=FML_function_block; Status.ID:=FML_fhpp_plus_value_not_valid;
			RETURN;

	
		ELSE	// do nothing
			;	
		
	END_CASE
	
	iObject									:= iObject + 1;			// increment the counter variable for FHPP+ objects in FML_REF

END_FOR


// fill up the remaining BYTEs of 'FHPP_PLUS_DATA_OUT' with zero
WHILE iAddress <= 23 DO
	pFHPP_PLUS_DATA_OUT^[iAddress]			:= 0;
	iAddress								:= iAddress + 1;		// increment the counter variable for address of the pointer in increments of 1	
END_WHILE
 
// write the output data from intern data buffer ('FHPP_PLUS_DATA_OUT') to the bus (to controller)
IF FML_REF.Modbus THEN												// Modbus word swapping
	FHPP_PLUS_Target1[0]	:= FHPP_PLUS_DATA_OUT[1];
	FHPP_PLUS_Target1[1]	:= FHPP_PLUS_DATA_OUT[0];
	FHPP_PLUS_Target1[2]	:= FHPP_PLUS_DATA_OUT[3];
	FHPP_PLUS_Target1[3]	:= FHPP_PLUS_DATA_OUT[2];
	FHPP_PLUS_Target1[4]	:= FHPP_PLUS_DATA_OUT[5];
	FHPP_PLUS_Target1[5]	:= FHPP_PLUS_DATA_OUT[4];
	FHPP_PLUS_Target1[6]	:= FHPP_PLUS_DATA_OUT[7];
	FHPP_PLUS_Target1[7]	:= FHPP_PLUS_DATA_OUT[6];
	FHPP_PLUS_Target2[0]	:= FHPP_PLUS_DATA_OUT[9];
	FHPP_PLUS_Target2[1]	:= FHPP_PLUS_DATA_OUT[8];
	FHPP_PLUS_Target2[2]	:= FHPP_PLUS_DATA_OUT[11];
	FHPP_PLUS_Target2[3]	:= FHPP_PLUS_DATA_OUT[10];
	FHPP_PLUS_Target2[4]	:= FHPP_PLUS_DATA_OUT[13];
	FHPP_PLUS_Target2[5]	:= FHPP_PLUS_DATA_OUT[12];
	FHPP_PLUS_Target2[6]	:= FHPP_PLUS_DATA_OUT[15];
	FHPP_PLUS_Target2[7]	:= FHPP_PLUS_DATA_OUT[14];
	FHPP_PLUS_Target3[0]	:= FHPP_PLUS_DATA_OUT[17];
	FHPP_PLUS_Target3[1]	:= FHPP_PLUS_DATA_OUT[16];
	FHPP_PLUS_Target3[2]	:= FHPP_PLUS_DATA_OUT[19];
	FHPP_PLUS_Target3[3]	:= FHPP_PLUS_DATA_OUT[18];
	FHPP_PLUS_Target3[4]	:= FHPP_PLUS_DATA_OUT[21];
	FHPP_PLUS_Target3[5]	:= FHPP_PLUS_DATA_OUT[20];
	FHPP_PLUS_Target3[6]	:= FHPP_PLUS_DATA_OUT[23];
	FHPP_PLUS_Target3[7]	:= FHPP_PLUS_DATA_OUT[22];
		
ELSE																// normal fieldbus: copy only
	pDataArray				:= ADR(FHPP_PLUS_DATA_OUT[0]);
	FHPP_PLUS_Target1		:= pDataArray^;
	pDataArray				:= ADR(FHPP_PLUS_DATA_OUT[8]);
	FHPP_PLUS_Target2		:= pDataArray^;
	pDataArray				:= ADR(FHPP_PLUS_DATA_OUT[16]);
	FHPP_PLUS_Target3		:= pDataArray^;
END_IF

Status.Err:=FALSE; Status.Cat:=FML_no_category; Status.ID:=FML_no_error;

(* ===== end of function block ============================= *)

END_FUNCTION_BLOCK

// Blocks/Parameterize/FPC_MULTI
(* ============================================================================
   FESTO AG & Co. KG, Esslingen - Copyright (c) 2015. All rights reserved.                       
 ------------------------------------------------------------------------------
 Functionblock:  PRM_MULTI  
 Description:    function block to pass an array of FHPP parameter to the motorcontroller
 Version:        V3.5.7.21         
 Composer:       bejk 
 Last Update:    13.11.2017                                                                           
----------------------------------------------------------------------------- *)
{library private}
(* ----------------------------------------------------------------------------
Date        Name                Activity                                                                              
01.04.2014  Benjamin Kilgus     V3.1: created
22.06.2015	Christian Hammer	adaptation to use this FB for all drives
25.09.2015  Christian Hammer	FPCC Modus in Step 1 changed (created device type)
13.11.2017	Christian Hammer	added SFC-DC and MTR-DCI controller
=============================================================================== *)
{library public}

(* use this function block only with the function blocks FML_Read and FML_Write *)


FUNCTION_BLOCK FPC_MULTI

VAR_IN_OUT
	FML_REF    		: DT_FML_REF;		// structure of the parameter to control and parametrize the motorcontroller
END_VAR

VAR_INPUT
	Execute     	: BOOL;            	// perfrom data exchange
	SizeOfParam 	: UINT;           	// size of the parameter array (Example : ARRAY [1..n] OF DT_FML_PRM_DESCRIPTION )
	AdrOfParam  	: POINTER TO BYTE; 	// 1. element of parameter array (Example : ARRAY [1..n] OF DT_FML_PRM_DESCRIPTION )
END_VAR

VAR_OUTPUT
	Done        	: BOOL;  			// transmission done
	Error			: BOOL; 			// transmission fault
	Status			: DT_FML_STATUS;	// structure with the status information of the function block	
	ParamNo     	: UINT;  			// progress of parameter transfer
END_VAR

{library private}
VAR
	bInit       	: BOOL	:=FALSE;						// status of inizialisation of the FB
	lMemberID   	: INT;									// local member ID of the FB		
	Step        	: INT 	:= 0;       					// step number of state machine 
	index       	: UINT;
	AnzParam    	: UINT;            						// calculated number of parameters
	iParamSize  	: UINT;           						// size of one parameter structure
	ptrParam   		: POINTER TO DT_FML_PRM_DESCRIPTION;  	// actual parameter
	
	TONInst			: TON;									// timer instance to monitor a timeout of the function block
	TimeStart		: BOOL;									// variable to start the timer instance
	TimeoutTime		: TIME := T#3S;							// timeout time 
	
	TimerFwBug		: TON;									// timer because of FW bug in SFC-Dc and MTR-DCI
	StartTimerFwBug	: BOOL;									// variable to start TimerFwBug	
END_VAR
{library public}

(* ====== initial block routine ===================================== *)
(* ----- get MemberID for this function block ------------------------*)
IF NOT bInit THEN
	FML_REF.MemberIDmax		:= FML_REF.MemberIDmax +1;
	lMemberID            	:= FML_REF.MemberIDmax;
	bInit              		:= TRUE;
	Status.Err:=FALSE; Status.Cat:=FML_function_block; Status.ID:=FML_init_active;
END_IF


(* ====== supervision of timeout ==================================== *)
(* ----- timer to monitor a timeout of the function block ------------*)
TimerFwBug(IN:= StartTimerFwBug, PT:= T#250MS);
TONInst(IN := TimeStart, PT := TimeoutTime);
IF TONInst.Q THEN
	Status.Err:=TRUE; Status.Cat:=FML_function_block; Status.ID:=FML_fb_timeout;
	Done					:= TRUE;
	Step					:= 30;
END_IF	


(* ===== logic part ================================================= *)

IF NOT Execute AND (Step <> 0) THEN
	FML_REF.MemberID		:= 0;
	FML_REF.ReqID			:= FML_FPC_REQ_none;
	FML_REF.PNU				:= 0;
	FML_REF.Subindex		:= 0;
	FML_REF.Value			:= 0;
	Step					:= 0;
END_IF

CASE Step OF
	0:(* initial prepare*)
		Done				:= FALSE;
  		ParamNo				:= 0;
		TimeStart			:= FALSE;
  		Status.Err:=FALSE; Status.Cat:=FML_no_category; Status.ID:=FML_no_error;

		IF Execute THEN
			iParamSize				:= SIZEOF(DT_FML_PRM_DESCRIPTION);
    		AnzParam                := (SizeOfParam) / iParamSize; 		// 12;
			// pointer not correct
			IF  SizeOfParam = 0 OR AdrOfParam = 0 THEN
				Status.Err:=TRUE; Status.Cat:=FML_function_block; Status.ID:=FML_pointer_to_zero;				// no input on either SizeOf or address of parameter
				Step					:= 30;
			// size of parameter not correct
			ELSIF (SizeOfParam MOD 16) <> 0 THEN
				Status.Err:=TRUE; Status.Cat:=FML_function_block; Status.ID:=FML_pointer_wrong_size;			// wrong size of parameter size has to by n*Size of DT_FML_PRM_DESCRIPTION
				Step					:= 30;
			// everything o.k. start task 
			ELSIF FML_REF.MemberID = 0 THEN
				FML_REF.MemberID    	:= lMemberID;
				FML_REF.ReqID          	:= FML_FPC_REQ_none;
				FML_REF.PNU            	:= 0;
				FML_REF.Subindex       	:= 0;
				FML_REF.Value			:= 0;
				index                   := 1;
				step                    := 1;
				Status.Err:=FALSE; Status.Cat:=FML_function_block; Status.ID:=FML_fb_busy;		
			// other FB active 
			ELSIF FML_REF.MemberID <> lMemberId THEN
				Status.Err:=FALSE; Status.Cat:=FML_function_block; Status.ID:=FML_other_fb_active;	
			END_IF		
		  END_IF
  
	1:(* set pointer to the paramter [i] *)
		TimeStart					:= TRUE; 
		IF NOT FML_REF.Done THEN
			TimeStart				:= FALSE;
			ptrParam 				:= AdrOfParam +  iParamSize * (index -1); 
		  	FML_REF.PNU				:= ptrParam^.PNU;
    	  	FML_REF.Subindex		:= ptrParam^.SUBINDEX;
		  
		  
			IF (FML_REF.DeviceType = CMMP_AS) 
			OR (FML_REF.DeviceType = CMMS_AS) 
			OR (FML_REF.DeviceType = CMMS_ST)
			OR (FML_REF.DeviceType = CMMD_AS) 
			OR (FML_REF.DeviceType = SFC_DC) 
			OR (FML_REF.DeviceType = MTR_DCI) THEN					(* CMMP-AS or CMMS_AS or CMMS_ST or CMMD_AS or SFC_DC or MTR_DCI *)					
				CASE ptrParam^.ACCESS OF
					(* read objekt *)
					0:(* 0 = PNU_11BIT *)
						FML_REF.FPCC_Modus	:= E_FML_FPC_MODUS.FML_FPC_MODUS_PNU_11BIT;
						FML_REF.ReqID		:= FML_FPC_REQ_read_array;
						IF FML_REF.DeviceType = SFC_DC OR FML_REF.DeviceType = MTR_DCI THEN				(* SFC-DC or MTR-DCI *)
							Step			:= 19;
						ELSE																			(* CMMP-AS or CMMS-AS or CMMS-ST or EMCA-EC or CMMO-ST *)
							Step			:= 20;	
						END_IF
							
					(* write object *)
					1:(* 1 = PNU_11BIT *)
						FML_REF.FPCC_Modus	:= E_FML_FPC_MODUS.FML_FPC_MODUS_PNU_11BIT;
						FML_REF.ReqID		:= FML_FPC_REQ_write_array_dword;
						FML_REF.DatatypeWR	:= ptrParam^.Length;
						FML_REF.Value		:= ptrParam^.VALUE;
						IF FML_REF.DeviceType = SFC_DC OR FML_REF.DeviceType = MTR_DCI THEN				(* SFC-DC or MTR-DCI *)
							Step			:= 9;
						ELSE																			(* CMMP-AS or CMMS-AS or CMMS-ST or EMCA-EC or CMMO-ST *)
							Step			:= 10;	
						END_IF
					
				ELSE
					Status.Err:=TRUE; Status.Cat:=FML_function_block; Status.ID:=FML_wrong_access_value;
					Step					:= 30;
				END_CASE
			
				
			ELSE 												(* CMMO-ST AND EMCA-EC *)
				CASE ptrParam^.ACCESS OF
					
					(* read objekt *)
					0,10:(* 0,10 = PNU_16BIT *)
						FML_REF.FPCC_Modus	:= E_FML_FPC_MODUS.FML_FPC_MODUS_PNU_16BIT;
						FML_REF.ReqID		:= FML_FPC_REQ_read_array;
						Step				:= 20; 
					(* write object *)
					1,11:(* 1,11 = PNU_16BIT *)
						FML_REF.FPCC_Modus	:= E_FML_FPC_MODUS.FML_FPC_MODUS_PNU_16BIT;
						FML_REF.ReqID		:= FML_FPC_REQ_write_array_dword;
						FML_REF.Value		:= ptrParam^.VALUE;
						Step				:= 10; // Write parameter
					
					(* read objekt *)
					20,30:(* 20 = data object, 30 = CAN object *)
						FML_REF.FPCC_Modus	:= ptrParam^.ACCESS / 10;
						FML_REF.ReqID		:= FML_FPC_REQ_read_array;
						Step				:= 20; 
						
					(* write object *)
					21,31:(* 21 = data object, 31 = CAN object *)
						FML_REF.FPCC_Modus	:= (ptrParam^.ACCESS -1) / 10;
						FML_REF.ReqID		:= FML_FPC_REQ_write_array_dword;
						FML_REF.Value		:= ptrParam^.VALUE;
						Step				:= 10; // Write parameter
						
				ELSE
					Status.Err:=TRUE; Status.Cat:=FML_function_block; Status.ID:=FML_wrong_access_value;
					Step					:= 30;
	 			END_CASE
			END_IF	
  		END_IF

	9:	(* delay state because of FW bug from SFC-DC and MTR-DCI *)
		StartTimerFwBug				:= TRUE;	
		IF TimerFwBug.Q THEN
			StartTimerFwBug			:= FALSE;
			step 					:= 10;
		END_IF	
		
	10:(* writing done *)
		TimeStart					:= TRUE; 
	  	ParamNo						:= index;
		
	  	IF FML_REF.Done AND NOT FML_REF.Err THEN
			TimeStart				:= FALSE;
			FML_REF.ReqID			:= FML_FPC_REQ_none;
			index					:= index + 1;
			IF FML_REF.DeviceType = SFC_DC OR FML_REF.DeviceType = MTR_DCI THEN				(* SFC-DC or MTR-DCI *)
				Step				:= 11;
			ELSE																			(* CMMP-AS or CMMS-AS or CMMS-ST or EMCA-EC or CMMO-ST *)
				Step				:= 1;	
			END_IF
			IF index > AnzParam THEN
		 		Done				:= TRUE;
		  		Status.Err:=FALSE; Status.Cat:=FML_no_category; Status.ID:=FML_no_error;
		  		Step				:= 30;
			END_IF;
	  	ELSIF FML_REF.Done AND FML_REF.Err THEN
			Done					:= TRUE;
			TimeStart				:= FALSE; 
			Status.Err:=TRUE; Status.Cat:=FML_parameter_transfer; Status.ID:=FML_REF.ActValue;
			Step					:= 30;
	  	END_IF;	

	11:	(* delay state because of FW bug from SFC-DC and MTR-DCI *)
		StartTimerFwBug				:= TRUE;	
		IF TimerFwBug.Q THEN
			StartTimerFwBug			:= FALSE;
			step 					:= 1;
		END_IF	
		
	19:	(* delay state because of FW bug from SFC-DC and MTR-DCI *)
		StartTimerFwBug				:= TRUE;	
		IF TimerFwBug.Q THEN
			StartTimerFwBug			:= FALSE;
			step 					:= 20;
		END_IF	
		
	20:(* reading done *)
		TimeStart					:= TRUE; 
  		ParamNo						:= index;
  		IF FML_REF.Done AND NOT FML_REF.Err THEN
			TimeStart				:= FALSE;
			FML_REF.ReqID			:= FML_FPC_REQ_none;
			ptrParam^.Length		:= FML_REF.DatatypeRD;
    		ptrParam^.VALUE			:= FML_REF.ActValue;
			index					:= index + 1;
    		IF FML_REF.DeviceType = SFC_DC OR FML_REF.DeviceType = MTR_DCI THEN				(* SFC-DC or MTR-DCI *)
				Step				:= 21;
			ELSE																			(* CMMP-AS or CMMS-AS or CMMS-ST or EMCA-EC or CMMO-ST *)
				Step				:= 1;	
			END_IF
   			IF index > AnzParam THEN
				Done      			:= TRUE;
				Status.Err:=FALSE; Status.Cat:=FML_no_category; Status.ID:=FML_no_error;
				Step				:= 30;
    			END_IF;
		ELSIF FML_REF.Done AND FML_REF.Err THEN
			Done					:= TRUE;
			TimeStart				:= FALSE;
			Status.Err:=TRUE; Status.Cat:=FML_parameter_transfer; Status.ID:=FML_REF.ActValue;
			Step					:= 30;
		END_IF

	21:	(* delay state because of FW bug from SFC-DC and MTR-DCI *)
		StartTimerFwBug				:= TRUE;	
		IF TimerFwBug.Q THEN
			StartTimerFwBug			:= FALSE;
			step 					:= 1;
		END_IF	
		
	30: (* done - do nothing *)
		;
END_CASE

Status.Msg				:= GetStatusMessage(Status);
Error					:= Status.Err;

(* ===== end of function block ============================= *)

END_FUNCTION_BLOCK

// Blocks/Parameterize/FPC_PNU
(* ============================================================================
   FESTO AG & Co. KG, Esslingen - Copyright (c) 2015. All rights reserved.                       

 Functionblock:  FPC_PNU  
 Description:    function block to pass single parameters to the motorcontroller
 Version:        V3.5.7.21         
 Composer:       bejk
 Last update:    13.11.2017                                                                           
------------------------------------------------------------------------------- *)
{library private}
(* ----------------------------------------------------------------------------
Date       Name             	Activity                                                                              
01.04.2014 Benjamin Kilgus  	V3.1  created out of CMMS_AS_PRM_SINGLE
06.02.2015 Rudolf Schenke   	UpperLimit/LowerLimit removed
                            	Change to fix 16-bit mode
                            	Reduce VISU to reduced module capabilities  
09.02.2015  Rudolf Schenke  	Implement 16-bit mode with hide preset 
22.06.2015	Christian Hammer	adaptation to use this FB for all drives
13.11.2017	Christian Hammer	added SFC-DC and MTR-DCI controller	
=============================================================================== *)
{library public}

(* use this function block only with the function blocks FML_Read and FML_Write *)

FUNCTION_BLOCK FPC_PNU

VAR_IN_OUT
	FML_REF				: DT_FML_REF;		// structure of the parameter to control and parametrize the motorcontroller
END_VAR

VAR_INPUT
	Execute				: BOOL;  			// perfrom data exchange
	Write				: BOOL;  			// read or write the parameter
	PNU					: INT;  			// number of the parameter to exchange
	Subindex			: INT; 				// subindex of the parameter to exchange
	Value				: DINT;  			// value of the parameter to exchange
	DatatypeWR          : USINT; 			// length of the parameter to exchange in byte (only necessary for SFC-DC and MTR-DCI)
END_VAR

VAR_OUTPUT
	Done				: BOOL;  			// execution done
	Error				: BOOL; 			// transmission fault
	Status				: DT_FML_STATUS;	// structure with the status information of the function block and FPC	
	ActPNU				: INT;  			// actual number of the parameter
	ActSubindex			: INT; 				// actual subindex of the parameter
	ActValue			: DINT;  			// read value of parameter
	DatatypeRD          : USINT; 			// actual length of the parameter in byte
END_VAR

{library private}
VAR
	bInit           	: BOOL	:=FALSE;	// status of inizialisation of the FB
	lMemberID   		: INT;				// local member ID of the FB
	
	TONInst				: TON;				// timer instance to monitor a timeout of the function block
	TimeStart			: BOOL;				// variable to start the timer instance
	TimeoutTime			: TIME := T#3S;		// timeout time 
END_VAR
{library public}

(* ====== initial block routine ===================================== *)
(* ----- get MemberID for this function block ------------------------*)
IF NOT bInit THEN
	FML_REF.MemberIDmax		:= FML_REF.MemberIDmax +1;
	lMemberID            	:= FML_REF.MemberIDmax;
	bInit              		:= TRUE;
	Status.Err:=FALSE; Status.Cat:=FML_function_block; Status.ID:=FML_init_active;
END_IF


(* ====== supervision of timeout ==================================== *)
(* ----- timer to monitor a timeout of the function block ------------*)
TONInst(IN := TimeStart, PT := TimeoutTime);
IF TONInst.Q THEN
	Done					:= TRUE;
	Status.Err:=TRUE; Status.Cat:=FML_function_block; Status.ID:=FML_fb_timeout;
END_IF		
	

(* ===== logic part ================================================= *)
(* ----- ASSIGNMENT OF STATUS --------------------------------------- *)
IF FML_REF.MemberID = lMemberId THEN
	IF FML_REF.Done AND NOT Status.Err THEN
 		TimeStart			:= FALSE;
		Done				:= TRUE;
		ActSubindex			:= DINT_TO_INT(FML_REF.ActSubindex);
		ActPNU				:= FML_REF.ActPNU;
		ActValue			:= FML_REF.ActValue;
		DatatypeRD      	:= FML_REF.DatatypeRD;
		Status.Err:=FALSE; Status.Cat:=FML_no_category; Status.ID:=FML_no_error;
		
		IF FML_REF.Err THEN
			Status.Err:=TRUE; Status.Cat:=FML_parameter_transfer; Status.ID:=FML_REF.ActValue;
		END_IF
	END_IF
END_IF

(* ----- ASSIGNMENT OF CONTROL at rising edge of execute ----------- *)
IF (FML_REF.MemberID = 0) AND Execute THEN
	TimeStart				:= TRUE;
	Status.Err:=FALSE; Status.Cat:=FML_function_block; Status.ID:=FML_fb_busy;
	FML_REF.MemberID		:= lMemberID;

	FML_REF.PNU          	:= PNU;
	FML_REF.Subindex     	:= Subindex;
	FML_REF.Value 			:= Value;

	IF Write THEN   		// write parameter
		FML_REF.DatatypeWR	:= DatatypeWR;
		FML_REF.ReqID		:= FML_FPC_REQ_write_array_dword;
	ELSE            		// read parameter
		FML_REF.ReqID		:= FML_FPC_REQ_read_array;	  
	END_IF
  	
	IF ((FML_REF.DeviceType = CMMP_AS) 
		OR (FML_REF.DeviceType = CMMS_AS) 
		OR (FML_REF.DeviceType = CMMS_ST))
		OR (FML_REF.DeviceType = CMMD_AS) 
		OR (FML_REF.DeviceType = SFC_DC) 
		OR (FML_REF.DeviceType = MTR_DCI) THEN					(* CMMP-AS or CMMS_AS or CMMS_ST or CMMD_AS or SFC_DC or MTR_DCI *)	
		FML_REF.FPCC_Modus	:= E_FML_FPC_MODUS.FML_FPC_MODUS_PNU_11BIT;
	ELSE 													(* CMMO-ST AND EMCA-EC *)
		FML_REF.FPCC_Modus := E_FML_FPC_MODUS.FML_FPC_MODUS_PNU_16BIT;
	END_IF
	
ELSIF (FML_REF.MemberID = lMemberId) AND NOT Execute THEN
	FML_REF.ReqID			:= FML_FPC_REQ_none;
	FML_REF.FPCC_Modus		:= 0;
	FML_REF.PNU				:= 0;
	FML_REF.Subindex		:= 0;
	FML_REF.Value			:= 0;
	ActSubindex				:= 0;
	ActPNU					:= 0;
	ActValue				:= 0;
	//TimeStart				:= TRUE;			(* BUG IN FIRMWARE CMMP_AS (V4.0.10.1501.13.61) --> Zeile in Lib derzeit nicht umsetzbar --> Problem am 14.09.2015 gemeldet (CHMM) *)
	IF NOT FML_REF.Done THEN
    	FML_REF.MemberID	:= 0;     						// free the modul after all transmission
		TimeStart			:= FALSE;
		Done				:= FALSE;
    	Status.Err:=FALSE; Status.Cat:=FML_no_category; Status.ID:=FML_no_error;
  	END_IF;

ELSIF (FML_REF.MemberID <> lMemberId) THEN
	IF Execute THEN
		Status.Err:=FALSE; Status.Cat:=FML_function_block; Status.ID:=FML_other_fb_active;
	ELSE
		Status.Err:=FALSE; Status.Cat:=FML_no_category; Status.ID:=FML_no_error;
	END_IF 
END_IF

Status.Msg					:= GetStatusMessage(Status);
Error						:= Status.Err;

(* ===== end of function block ============================= *)

END_FUNCTION_BLOCK

// Blocks/FHPP_CTRL
(* =====================================================================
   FESTO AG & Co. KG, Esslingen - Copyright 2015. All rights reserved.                       
 -----------------------------------------------------------------------
 Functionblock:  FHPP_CTRL  
 Description:    function block to control the motorcontroller
 Version:        V 3.5.4.5        
 Composer:       bejk 
 Last Update:    25.09.2015                                                                           
------------------------------------------------------------------------------- *)
{library private}
(* ----------------------------------------------------------------------------
Date        Name            	Activity                                                                              
01.04.2014  Benjamin Kilgus 	created (V3.0)
13.09.2014  Rudolf Schenke  	Redundant BOOL block replaced
14.11.2014  Rudolf Schenke  	Modbus swapping integrated
08.02.2015  Rudolf Schenke  	Force mode: Velocity limited to 100%
22.06.2015	Christian Hammer	adaptation to use this FB for all drives
25.09.2015	Christian Hammer	DragError in FollowingError renamed
29.02.2016	Christian Hammer	changed typecast of ActValue1 from BYTE into SINT
=============================================================================== *)
{library public}

(* use this function block only with the function blocks FML_Read and FML_Write *)

FUNCTION_BLOCK FHPP_CTRL

VAR_IN_OUT
	FML_REF		: DT_FML_REF;			// structure of the parameter to control and parametrize the motorcontroller
END_VAR

VAR_INPUT
	EnableDrive             : BOOL;		// CCON.0: drive enable
	Stop                    : BOOL;		// CCON.1: stop active == 0 / stop not active == 1
	Brake                   : BOOL;		// CCON.2: release brake
	ResetFault              : BOOL;		// CCON.3: quit active fault
	HMIAccessLocked         : BOOL;		// CCON.5: PLC control == 1 / HMI control == 0

	OPM                     : INT;		// operation mode

	Halt                    : BOOL;		// CPOS.0: Halt active == 0 / Halt not active == 1
	StartTask               : BOOL;		// CPOS.1: starts positioning task
	StartHoming             : BOOL;		// CPOS.2: starts homing task
	JoggingPos              : BOOL;		// CPOS.3 :jogging positive direction
	JoggingNeg              : BOOL;		// CPOS.4: jogging negative direction
	TeachActualValue        : BOOL;		// CPOS.5: teach actual position to selected record number
	ClearRemainingPosition  : BOOL;		// CPOS.6: clear remaining position if halt is/was active

	Relative        		: BOOL;		// CDIR.0: absolute = 0 / relative = 1
	DeactivateStrokeLimit   : BOOL;		// CDIR.5: If TRUE, stroke limit is deactivated (directmode/forcecontrol)
	
	RecordNo                : INT;		// set value of record number (recordmode)

	SetValueVelocity        : BYTE;		// set value velocity (directmode/positionmode
	SetValuePosition        : DINT;		// set value position (directmode/positioncontrol)
	SetValueForceRamp		: BYTE;		// set value for force-ramp
	SetValueForce           : DINT;		// set value force (directmode/forcecontrol)
	SetValueRotRamp         : BYTE;		// set value for rotation-speed-ramp (directmode/rotation-speed-control)
	SetValueRotSpeed        : DINT;		// set value for rotation-speed (directmode/rotation-speed-control)
	
	ExecuteFunction			: BOOL;		// execute cam disc function (TRUE = executed)
	SetFunctionNumber		: INT;		// set cam disc function number
	SetFunctionGroup		: INT;		// set cam disc function group
END_VAR

VAR_OUTPUT
	OPMString               : STRING;	// description of the operating mode
	StateOPMString          : STRING;	// description of the actual state

	DriveEnabled            : BOOL;		// SCON.0: 0 == disable, 1 == enable
	Ready                   : BOOL;		// SCON.1: drive is ready
	Warning                 : BOOL;		// SCON.2: indicates information to user (no stop of member)
	Fault                   : BOOL;		// SCON.3: indicates information to user (stop of member)
	SupplyVoltagePresent    : BOOL;		// SCON.4: 0 == not present, 1 == present
	ControlFCT_HMI          : BOOL;		// SCON.5: 0 == access MMI, 1 == PLC

	StateOPM                : INT;		// state of operation mode (INT)

	HaltActive              : BOOL;		// SPOS.0: 1 == halt is not active
	AckStart                : BOOL;		// SPOS.1: acknowledge start
	MC                      : BOOL;		// SPOS.2: motion complete
	AckTeach                : BOOL;		// SPOS.3: acknowledge teach
	DriveIsMoving           : BOOL;		// SPOS.4: 1 == drive is moving
	FollowingError          : BOOL;		// SPOS.5: 1 == drag error active
	StandstillControl       : BOOL;		// SPOS.6: 1 == Member is outside tolerance window after MC
	HomingValid       		: BOOL;		// SPOS.7: homing is valid
	
	VelocityLimitReached    : BOOL;		// SDIR.4: velocity limit reached (directmode/forcecontrol)
	StrokeLimitReached      : BOOL;		// SDIR.5: stroke limit reached (directmode/forcecontrol)

	RC1                     : BOOL;		// RSB.0: record chain condition 1 reached
	RCC                     : BOOL;		// RSB.1: record chain condition complete

	ActualRecordNo          : INT;		// actual record number (recordmode)*)
	ActualPosition          : DINT;		// actual position (directmode/positioncontrol)
	ActualVelocity          : DINT;		// actual velocity (directmode)
	ActualForce             : DINT;		// actual force (directmode/forcecontrol)
	ActualRotRamp           : DINT;		// actual value for rotation-speed-ramp (directmode/rotation-speed-control)
	ActualRotSpeed          : DINT;		// actual value for rotation-speed (directmode/rotation-speed-control)
	
	FunctionIsActive		: BOOL;		// status of cam disc function (TRUE = executed)
	ActualFunctionNumber	: INT;		// actual cam disc function number
	ActualFunctionGroup		: INT;		// actual cam disc function group	
END_VAR

VAR
	tempVisuMode			: INT;		// temporarily variable for visualization only
END_VAR	

{library private}

(*------------------------------------------------------*)
(* assignment of input data							  	*)
(*------------------------------------------------------*)

//assign SCON-Data
DriveEnabled		:= FML_REF.FHPP.IN.SCON.ENABLED;
Ready				:= FML_REF.FHPP.IN.SCON.OPEN;
Warning				:= FML_REF.FHPP.IN.SCON.WARN;
Fault				:= FML_REF.FHPP.IN.SCON.FAULT;
SupplyVoltagePresent:= FML_REF.FHPP.IN.SCON.VLOAD;
ControlFCT_HMI		:= FML_REF.FHPP.IN.SCON.FCT;

//assign SPOS-Data
HaltActive			:= FML_REF.FHPP.IN.SPOS.HALT;
AckStart			:= FML_REF.FHPP.IN.SPOS.ACK;
MC					:= FML_REF.FHPP.IN.SPOS.MC;
AckTeach			:= FML_REF.FHPP.IN.SPOS.TEACH;
DriveIsMoving		:= FML_REF.FHPP.IN.SPOS.MOV;
FollowingError		:= FML_REF.FHPP.IN.SPOS.DEV;
StandstillControl	:= FML_REF.FHPP.IN.SPOS.STILL;
HomingValid			:= FML_REF.FHPP.IN.SPOS.REF;

//assign Byte3-Data
IF FML_REF.FHPP.IN.SCON.OPM1 THEN	// ===== directmode active =====
	ActualRecordNo	:= 0;
	RC1				:= FALSE;
	RCC				:= FALSE;
	
	(* coding of operation mode state *)
	IF FML_REF.FHPP.IN.Byte3.7 AND (FML_REF.DeviceType=CMMP_AS) THEN // If the device is a CMMP-AS the cam disc function could be executed
		StateOPM.0 				:= FML_REF.FHPP.IN.SCON.OPM1; 		
		StateOPM.1 				:= FML_REF.FHPP.IN.SCON.OPM2;		
		StateOPM.2 				:= FML_REF.FHPP.IN.Byte3.1; 		// SDIR_B1: COM1
		StateOPM.3 				:= FML_REF.FHPP.IN.Byte3.2; 		// SDIR_B2: COM2
		
		ActualFunctionNumber.0	:= FML_REF.FHPP.IN.Byte3.3; 		// SDIR_B3: FNUM1
		ActualFunctionNumber.1	:= FML_REF.FHPP.IN.Byte3.4;			// SDIR_B3: FNUM2
		ActualFunctionGroup.0	:= FML_REF.FHPP.IN.Byte3.5;			// SDIR_B3: FGRP1
		ActualFunctionGroup.1	:= FML_REF.FHPP.IN.Byte3.6;			// SDIR_B3: FGRP2
		
		FunctionIsActive		:= TRUE;
		VelocityLimitReached	:= FALSE;
		StrokeLimitReached		:= FALSE;	
	ELSE															// cam disc function not executed
		StateOPM.0 				:= FML_REF.FHPP.IN.SCON.OPM1; 		
		StateOPM.1 				:= FML_REF.FHPP.IN.SCON.OPM2;		
		StateOPM.2 				:= FML_REF.FHPP.IN.Byte3.1; 		// SDIR_B1: COM1
		StateOPM.3 				:= FML_REF.FHPP.IN.Byte3.2; 		// SDIR_B2: COM2
		StateOPM.4 				:= FML_REF.FHPP.IN.Byte3.3; 		// SDIR_B3: FNUM1
		
		VelocityLimitReached	:= FML_REF.FHPP.IN.Byte3.4;			// SDIR_B3: FNUM2
		StrokeLimitReached		:= FML_REF.FHPP.IN.Byte3.5;			// SDIR_B3: FGRP1
		
		FunctionIsActive		:= FALSE;
		ActualFunctionNumber	:= 0;
		ActualFunctionGroup		:= 0;
	END_IF
	
ELSE								// ===== recordmode active =====              
	ActualRecordNo	:= BYTE_TO_USINT (FML_REF.FHPP.IN.Byte3);	// Byte_3 = record number
	RC1				:= FML_REF.FHPP.IN.ActValue1.0;
	RCC				:= FML_REF.FHPP.IN.ActValue1.1;	
	(* coding of operation mode state *)
	StateOPM.0 				:= FML_REF.FHPP.IN.SCON.OPM1;
	StateOPM.1 				:= FML_REF.FHPP.IN.SCON.OPM2;
	StateOPM.2 				:= 0;
	StateOPM.3 				:= 0;
	StateOPM.4 				:= 0;
	VelocityLimitReached	:= 0;
	StrokeLimitReached		:= 0;
	
	FunctionIsActive		:= FALSE;
	ActualFunctionNumber	:= 0;
	ActualFunctionGroup		:= 0;
END_IF


CASE StateOPM OF
	0:	(* recordmode *)
		ActualVelocity 		:= 0;
		ActualForce			:= 0;
		ActualRotRamp		:= 0;
		ActualRotSpeed		:= 0;
		ActualPosition		:= DWORD_TO_DINT(FML_REF.FHPP.IN.ActValue2);

	1:	(* directmode position control *)
		ActualVelocity 		:= SINT_TO_DINT(FML_REF.FHPP.IN.ActValue1);
		ActualForce			:= 0;
		ActualRotRamp		:= 0;
		ActualRotSpeed		:= 0;
		ActualPosition		:= DWORD_TO_DINT(FML_REF.FHPP.IN.ActValue2);
	
	5:  (* directmode force control *)
		ActualVelocity		:= 0;
		ActualForce			:= SINT_TO_DINT(FML_REF.FHPP.IN.ActValue1);
		ActualPosition		:= DWORD_TO_DINT(FML_REF.FHPP.IN.ActValue2);
		ActualRotRamp		:= 0;
		ActualRotSpeed		:= 0;	
	
	9:  (* directmode rotation-speed-control *)
		ActualVelocity		:= 0;
		ActualForce			:= 0;
		ActualRotRamp		:= SINT_TO_DINT(FML_REF.FHPP.IN.ActValue1);
 		ActualRotSpeed		:= DWORD_TO_DINT(FML_REF.FHPP.IN.ActValue2);
		ActualPosition		:= 0;
	
	ELSE
		ActualVelocity		:= 0;
		ActualForce			:= 0;
		ActualRotRamp		:= 0;
		ActualRotSpeed		:= 0;
		ActualPosition		:= 0;
END_CASE

StateOPMString := GetStateOPMString(StateOPM);		// specify state OPM string

(*------------------------------------------------------*)
(* assignment of output data						  	*)
(*------------------------------------------------------*)

OPMString	:= GetOPMString(OPM);   				// set the OPM string

//assign CCON-Data
FML_REF.FHPP.OUT.CCON.ENABLE	:= EnableDrive;
FML_REF.FHPP.OUT.CCON.STOP		:= Stop;
FML_REF.FHPP.OUT.CCON.BRAKE		:= Brake;
FML_REF.FHPP.OUT.CCON.RESET		:= ResetFault;
FML_REF.FHPP.OUT.CCON.res		:= FALSE;
FML_REF.FHPP.OUT.CCON.LOCK		:= HMIAccessLocked;
FML_REF.FHPP.OUT.CCON.OPM1		:= OPM.0; 			// former OperationModeB1;
FML_REF.FHPP.OUT.CCON.OPM2		:= OPM.1; 			// former OperationModeB2;

//assign CPOS-data
FML_REF.FHPP.OUT.CPOS.HALT		:= Halt;
FML_REF.FHPP.OUT.CPOS.START		:= StartTask;
FML_REF.FHPP.OUT.CPOS.HOM		:= StartHoming;
FML_REF.FHPP.OUT.CPOS.JOGP		:= JoggingPos;
FML_REF.FHPP.OUT.CPOS.JOGN		:= JoggingNeg;
FML_REF.FHPP.OUT.CPOS.TEACH		:= TeachActualValue;
FML_REF.FHPP.OUT.CPOS.CLEAR		:= ClearRemainingPosition;
FML_REF.FHPP.OUT.CPOS.res		:= FALSE;

//assign byte3-data
IF OPM.0  THEN  // >>>>	directmode  <<<<
	FML_REF.FHPP.OUT.Byte3.0	:= Relative;					// CDIR_B0: ABS
	FML_REF.FHPP.OUT.Byte3.1	:= OPM.2; 						// CDIR_B1: former ControlModeB1;
	FML_REF.FHPP.OUT.Byte3.2	:= OPM.3; 						// CDIR_B2: former ControlModeB2;
	
	IF ExecuteFunction	AND (FML_REF.DeviceType=CMMP_AS) THEN	(* cam disc function executed *)
		FML_REF.FHPP.OUT.Byte3.3	:= SetFunctionNumber.0;		// CDIR_B3: FNUM1
		FML_REF.FHPP.OUT.Byte3.4	:= SetFunctionNumber.1;		// CDIR_B4: FNUM2
		FML_REF.FHPP.OUT.Byte3.5	:= SetFunctionGroup.0;		// CDIR_B5: FGRP1
		FML_REF.FHPP.OUT.Byte3.6	:= SetFunctionGroup.1;		// CDIR_B6: FGRP2
		FML_REF.FHPP.OUT.Byte3.7	:= TRUE;					// CDIR_B7: FUNC
		
	ELSE														(* cam disc function not executed *)
		FML_REF.FHPP.OUT.Byte3.3	:= FALSE;					// CDIR_B3: FNUM1
		FML_REF.FHPP.OUT.Byte3.4	:= FALSE;					// CDIR_B4: FNUM2
		FML_REF.FHPP.OUT.Byte3.5	:= DeactivateStrokeLimit;	// CDIR_B5: FGRP1
		FML_REF.FHPP.OUT.Byte3.6	:= FALSE;					// CDIR_B6: FGRP2
		FML_REF.FHPP.OUT.Byte3.7	:= FALSE;					// CDIR_B7: FUNC
	END_IF
	

ELSE            // >>> recordmode <<< 
	FML_REF.FHPP.OUT.Byte3 			:= INT_TO_BYTE(RecordNo); 	// byte 3 = record no.
END_IF

CASE OPM OF
	0:(* recordmode *)
		FML_REF.FHPP.OUT.SetValue1		:= 0;    				// byte 4 
		FML_REF.FHPP.OUT.SetValue2		:= 0;    				// byte 5...8
  	
	1: (* directmode position control *)
		FML_REF.FHPP.OUT.SetValue1		:= MIN(SetValueVelocity, 100);				// byte 4 (permissible range of value is 0 to 100)
  		FML_REF.FHPP.OUT.SetValue2		:= DINT_TO_DWORD(SetValuePosition);			// byte 5...8
  
	5:(* directmode force control *)
		IF (FML_REF.DeviceType = CMMP_AS) THEN										(* CMMP-AS *)
			FML_REF.FHPP.OUT.SetValue1	:= MIN(SetValueForceRamp, 100);				// byte 4 (permissible range of value is 0 to 100)
			tempVisuMode				:= 1;
			
		ELSIF (FML_REF.DeviceType = CMMO_ST) 
		   OR (FML_REF.DeviceType = EMCA_EC) THEN 									(* CMMO-ST and EMCA-EC *)
			FML_REF.FHPP.OUT.SetValue1	:= MIN(SetValueVelocity, 100);				// byte 4 (permissible range of value is 0 to 100)
			tempVisuMode				:= 2;
			
		ELSE																		(* CMMS_AS and CMMS_ST and CMMD_AS *)
			FML_REF.FHPP.OUT.SetValue1	:= 0;										// byte 4 not used in controller
			tempVisuMode				:= 0;
		END_IF	
				
		FML_REF.FHPP.OUT.SetValue2		:= DINT_TO_DWORD(SetValueForce);			// force w/o limitation
  
	9:(* directmode rotation-speed-control *)
		FML_REF.FHPP.OUT.SetValue1		:= MIN(SetValueRotRamp, 100);				// byte 4 (permissible range of value is 0 to 100)
		FML_REF.FHPP.OUT.SetValue2		:= DINT_TO_DWORD(SetValueRotSpeed);			// byte 5...8
		
	ELSE (* illegal OPM is selected *)
		FML_REF.FHPP.OUT.SetValue1		:= 0;										// byte 4
		FML_REF.FHPP.OUT.SetValue2		:= 0;										// byte 5...8
END_CASE

(* ===== end of function block ============================= *)

END_FUNCTION_BLOCK

// Internal/Blocks/GetStateOPMString
(* ===============================================================================
   FESTO AG & Co. KG, Esslingen - Copyright 2015. All rights reserved.                       
 ---------------------------------------------------------------------------------
 Functionblock:  GetStateOPMString 
 Description:    function to get discription of the activ OPM 
 Version:        V 1.0        
 Composer:       Benjamin Kilgus 
 Last Update:    10.04.2014                                                                          
------------------------------------------------------------------------------- *)
{library private}
(* ----------------------------------------------------------------------------
Date        Name            	Activity                                                                              
10.04.2014	Benjamin Kilgus     created
=============================================================================== *)
{library public}

FUNCTION GetStateOPMString : string
VAR_INPUT
  iState : INT;
END_VAR

(*-----------------------------------------------------------
     logic
------------------------------------------------------------*)

CASE iState OF
   0:  GetStateOPMString := 'Record Mode active';
   1:  GetStateOPMString := 'Directmode Positioncontrol active';
   5:  GetStateOPMString := 'Directmode Forcecontrol active';
   9:  GetStateOPMString := 'Directmode Velocitycontrol active';
  13:  GetStateOPMString := 'Directmode Positioncontrol Energy Optimized active';
  17:  GetStateOPMString := 'Continuousmode active';
ELSE
   GetStateOPMString := 'not specified';
END_CASE

(* ===== end of function ================================== *)

END_FUNCTION

// Internal/Blocks/GetOPMString
(* ===============================================================================
   FESTO AG & Co. KG, Esslingen - Copyright 2015. All rights reserved.                       
 ---------------------------------------------------------------------------------
 Functionblock:  GetOPMString
 Description:    function to get discription of the selected OPM 
 Version:        V 1.0        
 Composer:       Benjamin Kilgus 
 Last Update:    10.04.2014                                                                          
------------------------------------------------------------------------------- *)
{library private}
(* ----------------------------------------------------------------------------
Date        Name            	Activity                                                                              
10.04.2014	Benjamin Kilgus     created
=============================================================================== *)
{library public}

FUNCTION GetOPMString : string
VAR_INPUT
  iOPM : INT;
END_VAR
VAR
END_VAR

(*-----------------------------------------------------------
     logic
------------------------------------------------------------*)

CASE iOPM OF
  0:  GetOPMString := 'Record Mode selected';
  1:  GetOPMString := 'Directmode Positioncontrol selected';
  2:  GetOPMString := 'Commissioning selected';
  3:  GetOPMString := 'Parameter loading selected';
  5:  GetOPMString := 'Directmode Forcecontrol selected';
  9:  GetOPMString := 'Directmode Velocitycontrol selected';
  13: GetOPMString := 'Directmode Positioncontrol Energy Optimized selected';
  17: GetOPMString := 'Continuousmode selected';
ELSE
  GetOPMString := 'not specified';
END_CASE

(* ===== end of function ================================== *)

END_FUNCTION

// Blocks/Parameterize/FPC_DATA_OBJECT
(* ============================================================================
   FESTO AG  Co., Esslingen - Copyright (c) 2015. All rights reserved.                       
 ------------------------------------------------------------------------------
 Functionblock:  FPC_DATA_OBJECT  
 Description:    function block to pass internal data objects to the controller
 Version:        V3.5.4.4        
 Composer:       bejk
 Last Update:    13.11.2017                                                                           
 ------------------------------------------------------------------------------ *)
{library private}
(* ----------------------------------------------------------------------------
Date        Name                Activity                                                                              
02.02.2010  Benjamin Kilgus     created
02.07.2013  Rudolf Schenke      Busy state and some other value clear
22.06.2015	Christian Hammer	adaptation to use this FB for all drives
04.09.2015  Christian Hammer	error handling (deleted RETVAL, created Status)
29.02.2016	Christian Hammer	set outputs to zero if not execute
13.11.2017	Christian Hammer	added blockade of FB for SFC-DC and MTR-DCI controller
=============================================================================== *)
{library public}

(* use this function block only with the function blocks FML_Read and FML_Write *)

FUNCTION_BLOCK FPC_DATA_OBJECT

VAR_IN_OUT
	FML_REF				: DT_FML_REF;		// structure of the parameter to control and parametrize the motorcontroller
END_VAR

VAR_INPUT
	Execute				: BOOL;  			// perfrom data exchange
	Write				: BOOL;  			// read or write the parameter (1=write / 0=read)
	Object				: INT; 				// number of internal data object
	Subindex			: INT; 				// subindex of the parameter to exchange
	Value				: DINT; 			// set value of internal data objects
END_VAR
VAR_OUTPUT
	Done				: BOOL; 			// transmission done
	Error				: BOOL; 			// transmission fault
	Status				: DT_FML_STATUS;	// structure with the status information of the function block and FPC
	ActObject			: INT;				// actual number of internal data objects
	ActSubindex			: DINT; 			// actual subindex of the parameter
	ActValue			: DINT; 			// actual value of internal data objects	
END_VAR

{library private}
VAR
	bInit           	: BOOL	:=FALSE;	// status of inizialisation of the FB
	lMemberID   		: INT;				// local member ID of the FB
	Step				: INT	:= 0;		// step number of the state machine

	TONInst				: TON;				// timer instance to monitor a timeout of the function block
	TimeStart			: BOOL;				// variable to start the timer instance
	TimeoutTime			: TIME := T#3S;		// timeout time 			
END_VAR
{library public}

(* ====== initial block routine ===================================== *)
(* ----- get MemberID for this function block ------------------------*)

IF NOT bInit THEN
	FML_REF.MemberIDmax		:= FML_REF.MemberIDmax +1;
	lMemberID				:= FML_REF.MemberIDmax;
	bInit					:= TRUE;
	Status.Err:=FALSE; Status.Cat:=FML_function_block; Status.ID:=FML_init_active;
END_IF

	
(* ====== supervision of timeout ==================================== *)
(* ----- timer to monitor a timeout of the function block ------------*)
TONInst(IN := TimeStart, PT := TimeoutTime);
IF TONInst.Q THEN
	Status.Err:=TRUE; Status.Cat:=FML_function_block; Status.ID:=FML_fb_timeout;
	Done					:= TRUE;
	Step					:= 100;
END_IF		

// this function block is not usable with SFC-DC and MTR-DCI
IF Execute 
	AND	((FML_REF.DeviceType = SFC_DC)
	OR (FML_REF.DeviceType = MTR_DCI)) THEN
		Done				:= TRUE;
		Status.Err:=TRUE; Status.Cat:=FML_function_block; Status.ID:=FML_wrong_device;
		Step				:= 100;
END_IF

(* ===== logic part ================================================= *)

IF NOT Execute AND (Step <> 0) THEN
 	FML_REF.MemberID		:= 0;
	FML_REF.ReqID			:= FML_FPC_REQ_none;
	FML_REF.FPCC_Modus		:= 0;
	FML_REF.PNU				:= 0;
	FML_REF.Subindex		:= 0;
	FML_REF.Value			:= 0;
	ActObject				:= 0;
	ActSubindex				:= 0;	
	ActValue				:= 0;
			
	Step					:= 0;
END_IF;

CASE Step OF
	0:(* *)
		Done				:= FALSE;
		TimeStart			:= FALSE;
		Status.Err:=FALSE; Status.Cat:=FML_no_category; Status.ID:=FML_no_error;

		IF (FML_REF.MemberID = 0) AND Execute THEN
    		FML_REF.MemberID		:= lMemberID;
			FML_REF.ReqID			:= FML_FPC_REQ_none;	
			FML_REF.PNU				:= 0;
			FML_REF.Subindex		:= 0;
			FML_REF.Value			:= 0;
			Status.Err:=FALSE; Status.Cat:=FML_function_block; Status.ID:=FML_fb_busy;
			
			IF (FML_REF.DeviceType = CMMP_AS) 
			OR (FML_REF.DeviceType = CMMS_AS) 
			OR (FML_REF.DeviceType = CMMS_ST)
			OR (FML_REF.DeviceType = CMMD_AS) THEN					(* CMMP-AS or CMMS_AS or CMMS_ST or CMMD_AS *)
				FML_REF.FPCC_Modus	:= FML_FPC_MODUS_PNU_11BIT;		// FPC standard
				Step				:= 10;				
			ELSE 													(* CMMO-ST AND EMCA-EC *)
				FML_REF.FPCC_Modus	:= FML_FPC_MODUS_DATA_OBJECT;	// EPC access for internal data objects
				Step				:= 20;
			END_IF
			
		ELSIF (FML_REF.MemberID <> lMemberId) AND Execute THEN
			Status.Err:=FALSE; Status.Cat:=FML_function_block; Status.ID:=FML_other_fb_active;
		END_IF

(* CMMP-AS or CMMS_AS or CMMS_ST or CMMD_AS or SFC_DC or MTR_DCI *)		
	10:(* open tunnel access *)
		FML_REF.ReqID				:= FML_FPC_REQ_write_array_dword; 
		FML_REF.PNU					:= 80;
		FML_REF.Subindex			:= 1;
		FML_REF.Value				:= Object;
		TimeStart					:= TRUE;
		
		IF FML_REF.Done AND NOT FML_REF.Err THEN
			TimeStart				:= FALSE;
      		FML_REF.ReqID         	:= FML_FPC_REQ_none;  
      		Step                  	:= 11;
  		(* error occured *)
  		ELSIF FML_REF.Done AND FML_REF.Err THEN
			TimeStart				:= FALSE;      		
      		Step                 	:= 30;
 		END_IF


	11:(* access granted *)
		TimeStart					:= TRUE;
	
		IF NOT FML_REF.Done THEN
			TimeStart				:= FALSE;
			(* write internal data objects *)
			IF Write THEN
				FML_REF.ReqID			:= FML_FPC_REQ_write_array_dword; 
				FML_REF.PNU				:= 82;
				FML_REF.Subindex		:= 1;
				FML_REF.Value			:= Value;
				Step					:= 30;
    		(* read internal data objects *)
			ELSE
				FML_REF.ReqID			:= FML_FPC_REQ_read_array;	  
				FML_REF.PNU				:= 81;
				FML_REF.Subindex		:= 1;
				FML_REF.Value			:= 0;
				Step					:= 30;
			END_IF
		END_IF
		
(* CMMO-ST AND EMCA-EC *)
	20:		
		IF Write THEN
			FML_REF.ReqID			:= FML_FPC_REQ_write_array_dword; 
		ELSE
			FML_REF.ReqID			:= FML_FPC_REQ_read_array;
		END_IF	
			
		FML_REF.PNU					:= Object;
		FML_REF.Subindex			:= Subindex;
		FML_REF.Value				:= Value;
		Step						:= 30;

	30:(* set output variables *)
		TimeStart					:= TRUE;
		
		IF FML_REF.Done THEN
			FML_REF.ReqID			:= FML_FPC_REQ_none;
			TimeStart				:= FALSE;
			Done					:= TRUE;
			Step					:= 100;
			
			IF FML_REF.Err THEN
				Status.Err:=TRUE; Status.Cat:=FML_parameter_transfer; Status.ID:=FML_REF.ActValue;
				ActValue			:= 0;
				ActSubindex			:= 0;
				ActObject			:= 0;   
			ELSE
				Status.Err:=FALSE; Status.Cat:=FML_no_category; Status.ID:=FML_no_error;
				
				IF (FML_REF.DeviceType = CMMP_AS) 
				OR (FML_REF.DeviceType = CMMS_AS) 
				OR (FML_REF.DeviceType = CMMS_ST)
				OR (FML_REF.DeviceType = CMMD_AS) 
				OR (FML_REF.DeviceType = SFC_DC) 
				OR (FML_REF.DeviceType = MTR_DCI) THEN					(* CMMP-AS or CMMS_AS or CMMS_ST or CMMD_AS or SFC_DC or MTR_DCI *)
					ActObject			:= Object;
					ActSubindex			:= Subindex;
					ActValue			:= FML_REF.ActValue;			
				ELSE 												(* CMMO-ST AND EMCA-EC *)
					ActObject			:= FML_REF.ActPNU;
					ActSubindex			:= FML_REF.ActSubindex;
					ActValue			:= FML_REF.ActValue;
				END_IF
			END_IF
  		END_IF
	
	100: (* done - do nothing *)
		;
		
END_CASE

Status.Msg					:= GetStatusMessage(Status);
Error						:= Status.Err;

(* ===== end of function block ============================= *)

END_FUNCTION_BLOCK

// Blocks/Parameterize/FPC_DIAG
(* ============================================================================
   FESTO AG & Co. KG, Esslingen - Copyright (c) 2015. All rights reserved.                       

 Functionblock:  FPC_DIAG
 Description:    function block to read the most actual error
 Version:        V3.5.7.21         
 Composer:       bejk
 Date:           13.11.2017                                                                           
------------------------------------------------------------------------------- *)
{library private}
(* ----------------------------------------------------------------------------
Date        Name             	Activity                                                                              
01.04.2014  Benjamin Kilgus  	V3.1  created out of CMMS_AS_PRM_SINGLE
09.02.2015  Rudolf Schenke   	Implement 16-bit mode with hide preset
22.06.2015	Christian Hammer	adaptation to use this FB for all drives
04.09.2015  Christian Hammer	error handling (deleted RETVAL, created Status)
13.11.2017	Christian Hammer	added blockade of FB for SFC-DC and MTR-DCI controller
=============================================================================== *)
{library public}

(* use this function block only with the function blocks FML_Read and FML_Write *)

FUNCTION_BLOCK FPC_DIAG

VAR_IN_OUT
	FML_REF        		: DT_FML_REF;		// structure of the parameter to control and parametrize the motorcontroller
END_VAR

VAR_INPUT															
	Execute         	: BOOL;  			// perfrom data exchange
END_VAR

VAR_OUTPUT
	Done            	: BOOL;  			// execution done
	Error				: BOOL; 			// transmission fault
	Status				: DT_FML_STATUS;	// structure with the status information of the function block and FPC	
	MessageNumber   	: INT;  			// fault occured
	MessageDescription  : STRING;			// discription of the error
END_VAR

{library private}
VAR
	bInit           	: BOOL	:=FALSE;	// status of inizialisation of the FB
	lMemberID   		: INT;				// local member ID of the FB	
	
	TONInst				: TON;				// timer instance to monitor a timeout of the function block
	TimeStart			: BOOL;				// variable to start the timer instance
	TimeoutTime			: TIME := T#3S;		// timeout time 
END_VAR
{library public}

(* ====== initial block routine ===================================== *)
(* ----- get MemberID for this function block ------------------------*)
IF NOT bInit THEN
	FML_REF.MemberIDmax		:= FML_REF.MemberIDmax +1;
	lMemberID            	:= FML_REF.MemberIDmax;
	bInit              		:= TRUE;
	Status.Err:=FALSE; Status.Cat:=FML_function_block; Status.ID:=FML_init_active;
END_IF


(* ====== supervision of timeout ==================================== *)
(* ----- timer to monitor a timeout of the function block ------------*)
TONInst(IN := TimeStart, PT := TimeoutTime);
IF TONInst.Q THEN
	Done					:= TRUE;
	Status.Err:=TRUE; Status.Cat:=FML_function_block; Status.ID:=FML_fb_timeout;
END_IF					

	
(* ===== logic part ================================================= *)
(* ----- ASSIGNMENT OF STATUS --------------------------------------- *)
// this function block is not usable with SFC-DC and MTR-DCI
IF ((FML_REF.DeviceType = SFC_DC)
OR (FML_REF.DeviceType = MTR_DCI)) THEN
	IF Execute THEN
		Done					:= TRUE;
		Status.Err:=TRUE; Status.Cat:=FML_function_block; Status.ID:=FML_wrong_device;
	ELSE
		Done					:= FALSE;
		Status.Err:=FALSE; Status.Cat:=FML_no_category; Status.ID:=FML_no_error;
	END_IF
ELSE

	IF FML_REF.MemberID = lMemberId THEN
		IF FML_REF.Done AND NOT FML_REF.Err AND NOT Status.Err THEN
			Done              	:= TRUE;
			TimeStart			:= FALSE;
			
			IF FML_REF.ActValue = 65535 THEN 			// special: -1 to 0
				MessageNumber 	:= 0; 
			ELSE
				MessageNumber	:= DINT_TO_INT(FML_REF.ActValue);	
			END_IF  
			
			MessageDescription	:= FaultString(MessageNumber, FML_REF.DeviceType);
			Status.Err:=FALSE; Status.Cat:=FML_no_category; Status.ID:=FML_no_error;
			
		ELSIF FML_REF.Err THEN
			Status.Err:=TRUE; Status.Cat:=FML_parameter_transfer; Status.ID:=FML_REF.ActValue;
		END_IF
	END_IF
	
	(* ----- ASSIGNMENT OF CONTROL at rising edge of Execute ------------ *)
	IF (FML_REF.MemberID = 0) AND Execute THEN
		TimeStart				:= TRUE;
		Status.Err:=FALSE; Status.Cat:=FML_function_block; Status.ID:=FML_fb_busy;
		FML_REF.MemberID    	:= lMemberID;
		FML_REF.ReqID			:= FML_FPC_REQ_read_array;
	 
		IF (FML_REF.DeviceType = CMMP_AS) 
		OR (FML_REF.DeviceType = CMMS_AS) 
		OR (FML_REF.DeviceType = CMMS_ST)
		OR (FML_REF.DeviceType = CMMD_AS) THEN					(* CMMP-AS or CMMS_AS or CMMS_ST or CMMD_AS *)
			FML_REF.FPCC_Modus 	:= E_FML_FPC_MODUS.FML_FPC_MODUS_PNU_11BIT;
			FML_REF.PNU			:= 201;
			FML_REF.Subindex	:= 1;
	
		ELSE 													(*******EMCA-EC or CMMO-ST*******)	
			FML_REF.FPCC_Modus 	:= E_FML_FPC_MODUS.FML_FPC_MODUS_PNU_16BIT;
			FML_REF.PNU			:= 205;
			FML_REF.Subindex	:= 1;
		END_IF
		FML_REF.Value			:= 0;
	
	ELSIF (FML_REF.MemberID = lMemberId) AND NOT Execute THEN
		FML_REF.ReqID			:= FML_FPC_REQ_none;
		FML_REF.PNU				:= 0;
		FML_REF.Subindex		:= 0;
		FML_REF.Value			:= 0;
		MessageNumber			:= 0;
		MessageDescription		:= '';
		TimeStart				:= TRUE;
		IF NOT FML_REF.Done THEN
			FML_REF.MemberID	:= 0;     				// free the modul after all transmission
			TimeStart			:= FALSE;
			Done				:= FALSE;
			Status.Err:=FALSE; Status.Cat:=FML_no_category; Status.ID:=FML_no_error;
		END_IF;
		
	ELSIF (FML_REF.MemberID <> lMemberId) THEN
		IF Execute THEN
			Status.Err:=FALSE; Status.Cat:=FML_function_block; Status.ID:=FML_other_fb_active;
		ELSE
			Status.Err:=FALSE; Status.Cat:=FML_no_category; Status.ID:=FML_no_error;
		END_IF 
	END_IF
END_IF

Status.Msg						:= GetStatusMessage(Status);
Error							:= Status.Err;

(* ===== end of function block ============================= *)

END_FUNCTION_BLOCK

// Blocks/Parameterize/FPC_FILE_ARRAY
(* ============================================================================
   FESTO AG & Co. KG, Esslingen - Copyright 2015. All rights reserved.                       
 ------------------------------------------------------------------------------
 Functionblock: PRM_FILE_ARRAY
 Description:   function block to save and restore parameter file in a array
                  - Upload: from controller to PLC (array)
                  - Download: from PLC (array) to controller 
 ------------------------------------------------------------------------------
 Version:        V3.5.7.21         
 Composer:       bejk 
 Last Update:    13.11.2017                                                                               
 ------------------------------------------------------------------------------ *)
{library private}
(* ----------------------------------------------------------------------------
 Date       Name             	Activity                                                                              
 01.04.2014 Benjamin Kilgus  	created
 07.09.2014 Rudolf Schenke   	NextSequence() for Sequence++ created
                             	Correct all compiler warning causes 
                             	Set the fix directory name to 'CMMOparameter'
                             	Download: More direct buffer management
 14.09.2014 Rudolf Schenke   	VIS_CMMO_PRM_FILE prepared and adapted
 29.09.2014 Rudolf Schenke   	Redesign from file functions to file FBs
 10.12.2014 Rudolf Schenke   	Redesign der Schnittstelle zum file FB 
 14.01.2015 Rudolf Schenke   	Fehler bei Create Directory korrigiert (173989)
 09.03.2015 Rudolf Schenke   	CMMO_PRM_FILE: Umstellung auf neue IODD für IO-Link                              
 22.06.2015	Christian Hammer	adaptation to use this FB for all drives	
 29.02.2016	Christian Hammer	changed Line 265 (IF Status.ID==FML_par_file_err)
 20.10.2017 Christian Hammer	device type "CMMP_AS" added (deleted in line 12)
 13.11.2017	Christian Hammer	added blockade of FB for SFC-DC and MTR-DCI controller
=============================================================================== *)
{library public}

(* use this function block only with the function blocks FML_Read and FML_Write *)

FUNCTION_BLOCK FPC_FILE_ARRAY

VAR_IN_OUT
	FML_REF    		: DT_FML_REF;			// structure of the parameter to control and parametrize the motorcontroller
END_VAR

VAR_INPUT
	Execute     	: BOOL;     			// perform data exchange	
	Upload 			: BOOL;	    			// upload operation
	Download    	: BOOL;     			// download operation
	SizeOfFileArray : UINT;           		// size of the file array
	AdrOfFileArray  : POINTER TO BYTE; 		// 1. element of file array
END_VAR

VAR_OUTPUT
	Done        	: BOOL;  				// transmission done 
	Error			: BOOL; 				// error during execution	
	Status			: DT_FML_STATUS;		// structure with the status information of the function block	
	CountByte		: DINT;        			// dynamic byte counter
	FileSize		: DINT;	        		// resulting file size
END_VAR		

{library private}

VAR CONSTANT
 	udLength			: INT := 6;			// length of a file token
	ArrayWithZeros		: ARRAY[0..5] OF BYTE := [udLength(0)]; 			//[0,0,0,0,0,0]
END_VAR

VAR
	//general variables
	bInit      			: BOOL := FALSE;	// init flag
	lMemberID     		: INT;
	SendRepeat			: INT;
	Sequence			: INT;   			// sequence counter (incremented after each transfer)
	Step				: INT;      		// state machine

	//buffer
	pbyBuffer			: POINTER TO ARRAY [1..udLength] OF BYTE;
	Buffer				: ARRAY [1..udLength] OF BYTE := [udLength(0)]; 	//[0,0,0,0,0,0]
	PtrToDataFileArray  : POINTER TO BYTE;
	i					: INT;
		
	// visu
	vis_upload			: BOOL;   			// upload active for visu
	vis_download		: BOOL;  			// download active for visu

	//timout
	TimeStart			: BOOL;
	TimeStop			: BOOL;
 	TONInst				: TON;
END_VAR
{library public}

(* ====== initial block routine ===================================== *)
(* ----- get MemberID for this function block ------------------------*)
IF NOT bInit THEN
	FML_REF.MemberIDmax		:= FML_REF.MemberIDmax +1;
	lMemberID            	:= FML_REF.MemberIDmax;
	bInit              		:= TRUE;
	Status.Err:=FALSE; Status.Cat:=FML_function_block; Status.ID:=FML_init_active;
END_IF

//no file transfer in CMMS_AS or CMMS_ST or CMMD_AS
IF Execute 
	AND ((FML_REF.DeviceType = CMMS_AS) 
		OR (FML_REF.DeviceType = CMMS_ST)
		OR (FML_REF.DeviceType = CMMD_AS)
		OR (FML_REF.DeviceType = SFC_DC)
		OR (FML_REF.DeviceType = MTR_DCI)) THEN
			Done				:= TRUE;
			Status.Err:=TRUE; Status.Cat:=FML_function_block; Status.ID:=FML_wrong_device;
			Step				:= 27;
END_IF


(* ===== logic part ================================================= *)
IF NOT Execute AND (Step <> 0) THEN 										// reset all parameter (also bus data)
	FML_REF.MemberID     				:= 0;
	FML_REF.ReqID      	    			:= FML_FPC_REQ_none;
	FML_REF.FPCC_Modus					:= 0;
	FML_REF.FPCC_Packet.Control			:= 0;
	FML_REF.FPCC_Packet.BitSequenceNr	:= 0;
	FML_REF.FPCC_Packet.Data			:= ArrayWithZeros;
			
	Step 								:= 0;
END_IF

TONInst(IN := TimeStart, PT := T#3S, Q => TimeStop);						//timer for timeout


CASE Step OF 
	0:(* initial prepare*)
		Done			:= FALSE;
		Sequence		:= 0;
		CountByte 		:= 0;
		FileSize		:= 0;
		vis_download	:= FALSE;
		vis_upload		:= FALSE;
		SendRepeat		:= 0;
		Status.Err:=FALSE; Status.Cat:=FML_no_category; Status.ID:=FML_no_error;
    
		IF Execute AND FML_REF.MemberID = 0 THEN							// parameterchannel is free
			FML_REF.MemberID   		:= lMemberID;
			FML_REF.ReqID			:= FML_FPC_REQ_none;
					  
    		// check for double mode selection by visu
			IF NOT (Upload XOR Download) THEN  								// both or none are selected -> error
 				Status.Err:=TRUE; Status.Cat:=FML_parameter_transfer; Status.ID:=FML_direction_err;
				Step				:= 27;
       			RETURN;
			
			ELSIF Upload AND NOT Download THEN
				pbyBuffer			:= ADR(FML_REF.FPCS_Packet.Data);
				PtrToDataFileArray	:= AdrOfFileArray;
				vis_upload 			:= TRUE;
				Status.Err:=FALSE; Status.Cat:=FML_function_block; Status.ID:=FML_fb_busy;  	// execute starts here				
				Step 				:= 1;														// step 1 = starts upload
			
			ELSIF Download AND NOT Upload THEN
				pbyBuffer 	  		:= ADR(Buffer);
				PtrToDataFileArray	:= AdrOfFileArray;
				vis_download		:= TRUE;
				Status.Err:=FALSE; Status.Cat:=FML_function_block; Status.ID:=FML_fb_busy; 		// execute starts here
				Step 				:= 6;														// step 6 = starts download
			END_IF

	  	  // other FB active 
		ELSIF Execute AND FML_REF.MemberID <> lMemberId THEN
			Status.Err:=FALSE; Status.Cat:=FML_function_block; Status.ID:=FML_other_fb_active; 		
		END_IF
		
		
    //===== upload handling ===============
	1: (*start requirement - upload*)
		FML_REF.FPCC_Modus 			    	:= 4;							// choose mode
		FML_REF.ReqID 						:= FML_FPC_REQ_read_file; 		// upload
		FML_REF.FPCC_Packet.Control			:= FML_FPC_FILE_TRANSFER_start; // start transmission
		FML_REF.FPCC_Packet.BitSequenceNr	:= Sequence;
		FML_REF.FPCC_Packet.Data			:= Buffer; 						// user data are zero
		TimeStart 							:= TRUE; 						// start timer for timeout
		Step 								:= 2;
		
	2: (*wait for response from controller - upload*)
		// controller also sends upload data with the size of the parameter file
		IF FML_REF.RespID = FML_FPC_RESP_file_done AND FML_REF.FPCS_Packet.Control = FML_REF.FPCC_Packet.Control AND FML_REF.FPCS_Packet.BitSequenceNr = Sequence THEN
			Buffer							:= FML_REF.FPCS_Packet.Data;	// write incoming data from controller into buffer (6 Byte)
			FOR i := 0 TO 5 DO
				PtrToDataFileArray^			:= Buffer[i+1];					// write data from buffer to output (each byte separately)
				PtrToDataFileArray			:= PtrToDataFileArray + 1;
			END_FOR
			
			IF Sequence = 0 THEN 											// save size of parameterfile
				CalculateFilesize();  										// calculate size of file as a multiple of udLength	
				
				IF FileSize > SizeOfFileArray THEN							// check if the array is big enough
					Step 			    	:= 27; 							// array is to small --> error state
					Status.Err:=TRUE; Status.Cat:=FML_parameter_transfer; Status.ID:=FML_volume_err;
					RETURN;
				END_IF
			END_IF
		 	
			CountByte 						:= CountByte + udLength;		// count up the bytes
			NextSequence();													// count up the sequence
			TimeStart 						:= FALSE; 						// reset timer
			Step 							:= 3;
			
		ELSE //---- timeout ----
			IF TimeStop THEN
				TimeStart 					:= FALSE; 						// reset timer
				Step 						:= 4; 							// start acknowledgment is missing -->  check Step 4 on error
			END_IF
		END_IF

	3: (*request package - upload*)
		FML_REF.FPCC_Packet.Control 		:= FML_FPC_FILE_TRANSFER_active;
		FML_REF.FPCC_Packet.BitSequenceNr 	:= Sequence;
		FML_REF.FPCC_Packet.Data 			:= Buffer;		
		Step 								:= 4;

